KUKA KRL program: f1_Kuka_APT202T03S02.SRC

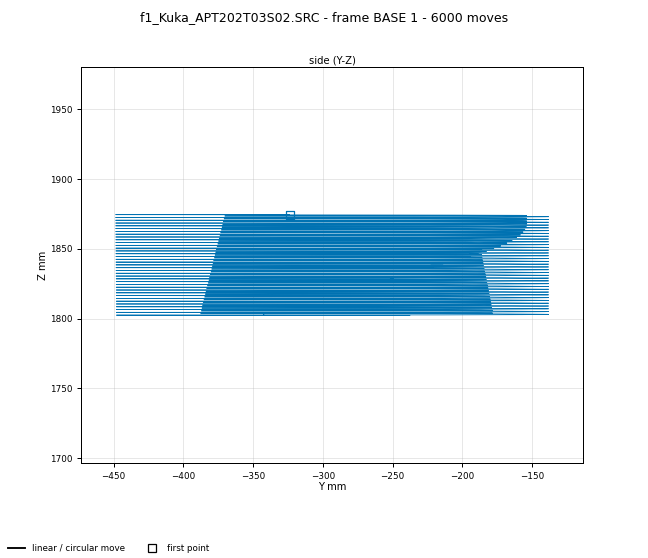
[picture p0: tool path of f1_Kuka_APT202T03S02.SRC in frame BASE 1, 6000 of 6001 moves have a stored position in this frame; points joined in program order, loops and branches not executed]
&ACCESS RVP
&REL 2
&PARAM TEMPLATE = C:\KRC\Roboter\Template\vorgabe
&PARAM EDITMASK = *
DEF f1_Kuka_APT202T03S02()


;FOLD INI;%{PE}%V3.2.0,%MKUKATPBASIS,%CINIT,%VCOMMON,%P
  ;FOLD BAS INI;%{E}%V3.2.0,%MKUKATPBASIS,%CINIT,%VINIT,%P
    GLOBAL INTERRUPT DECL 3 WHEN $STOPMESS==TRUE DO IR_STOPM ( )
    INTERRUPT ON 3
    BAS (#INITMOV,0 )
  ;ENDFOLD (BAS INI)
  ;FOLD USER INI;%{E}%V3.2.0,%MKUKATPUSER,%CINIT,%VINIT,%P
    ;Make your modifications here
  ;ENDFOLD (USER INI)
;ENDFOLD (INI)


;*** Make Null PTP Move
  PTP $pos_act

;*** Auto Load The Correct TOOL Data
  $tool=tool_data[3]

;*** Auto Load The Correct BASE Data
  $base=base_data[1]

  $ADVANCE = 5

;*** Restate Last Velocity
MMPM(30000.0)
SetRPM(6000)
LIN {X 0.160,Y -323.868,Z 1874.590,A 0.000,B 0.000,C 90.000,E1 106.260} C_DIS
LIN {X -0.109,Y -337.538,Z 1874.580,A 0.000,B 0.000,C 90.000,E1 104.411} C_DIS
LIN {X 0.038,Y -352.392,Z 1874.570,A 0.000,B 0.000,C 90.000,E1 102.535} C_DIS
LIN {X 0.047,Y -370.795,Z 1874.558,A 0.000,B 0.000,C 90.000,E1 100.489} C_DIS
LIN {X 0.119,Y -389.616,Z 1874.548,A 0.000,B 0.000,C 90.000,E1 98.624} C_DIS
LIN {X 0.014,Y -408.857,Z 1874.539,A 0.000,B 0.000,C 90.000,E1 96.947} C_DIS
LIN {X -0.177,Y -431.224,Z 1874.529,A 0.000,B 0.000,C 90.000,E1 95.220} C_DIS
LIN {X -0.017,Y -439.619,Z 1874.526,A 0.000,B 0.000,C 90.000,E1 94.588} C_DIS
LIN {X 0.199,Y -441.761,Z 1874.524,A 0.000,B 0.000,C 90.000,E1 94.359} C_DIS
LIN {X 0.089,Y -443.727,Z 1874.523,A 0.000,B 0.000,C 90.000,E1 94.131} C_DIS
LIN {X 0.009,Y -445.233,Z 1874.522,A 0.000,B 0.000,C 90.000,E1 93.898} C_DIS
LIN {X 0.189,Y -446.476,Z 1874.520,A 0.000,B 0.000,C 90.000,E1 93.612} C_DIS
LIN {X -0.075,Y -447.396,Z 1874.519,A 0.000,B 0.000,C 90.000,E1 93.383} C_DIS
LIN {X -0.118,Y -448.428,Z 1874.516,A 0.000,B 0.000,C 90.000,E1 92.865} C_DIS
LIN {X -0.177,Y -448.508,Z 1874.513,A 0.000,B 0.000,C 90.000,E1 92.350} C_DIS
LIN {X -0.213,Y -447.651,Z 1874.510,A 0.000,B 0.000,C 90.000,E1 91.833} C_DIS
LIN {X 0.183,Y -445.726,Z 1874.507,A 0.000,B 0.000,C 90.000,E1 91.260} C_DIS
LIN {X 0.128,Y -442.593,Z 1874.504,A 0.000,B 0.000,C 90.000,E1 90.745} C_DIS
LIN {X 0.008,Y -431.075,Z 1874.494,A 0.000,B 0.000,C 90.000,E1 88.912} C_DIS
LIN {X -0.023,Y -421.003,Z 1874.485,A 0.000,B 0.000,C 90.000,E1 87.306} C_DIS
LIN {X -0.120,Y -409.228,Z 1874.474,A 0.000,B 0.000,C 90.000,E1 85.412} C_DIS
LIN {X 0.015,Y -397.325,Z 1874.464,A 0.000,B 0.000,C 90.000,E1 83.451} C_DIS
LIN {X -0.090,Y -385.367,Z 1874.453,A 0.000,B 0.000,C 90.000,E1 81.489} C_DIS
LIN {X 0.040,Y -373.481,Z 1874.441,A 0.000,B 0.000,C 90.000,E1 79.454} C_DIS
LIN {X -0.066,Y -355.484,Z 1874.423,A 0.000,B 0.000,C 90.000,E1 76.228} C_DIS
LIN {X -0.066,Y -341.683,Z 1874.408,A 0.000,B 0.000,C 90.000,E1 73.504} C_DIS
LIN {X -0.122,Y -329.802,Z 1874.395,A 0.000,B 0.000,C 90.000,E1 71.040} C_DIS
LIN {X 0.107,Y -316.779,Z 1874.379,A 0.000,B 0.000,C 90.000,E1 68.156} C_DIS
LIN {X -0.103,Y -305.735,Z 1874.364,A 0.000,B 0.000,C 90.000,E1 65.613} C_DIS
LIN {X -0.074,Y -296.186,Z 1874.352,A 0.000,B 0.000,C 90.000,E1 63.307} C_DIS
LIN {X 0.124,Y -285.518,Z 1874.337,A 0.000,B 0.000,C 90.000,E1 60.589} C_DIS
LIN {X 0.126,Y -276.095,Z 1874.323,A 0.000,B 0.000,C 90.000,E1 58.201} C_DIS
LIN {X -0.021,Y -266.617,Z 1874.310,A 0.000,B 0.000,C 90.000,E1 55.801} C_DIS
LIN {X -0.060,Y -257.019,Z 1874.296,A 0.000,B 0.000,C 90.000,E1 53.336} C_DIS
LIN {X -0.008,Y -247.409,Z 1874.282,A 0.000,B 0.000,C 90.000,E1 50.803} C_DIS
LIN {X -0.043,Y -237.926,Z 1874.268,A 0.000,B 0.000,C 90.000,E1 48.243} C_DIS
LIN {X 0.069,Y -226.120,Z 1874.249,A 0.000,B 0.000,C 90.000,E1 44.838} C_DIS
LIN {X 0.023,Y -214.916,Z 1874.230,A 0.000,B 0.000,C 90.000,E1 41.391} C_DIS
LIN {X -0.011,Y -205.742,Z 1874.213,A 0.000,B 0.000,C 90.000,E1 38.257} C_DIS
LIN {X 0.104,Y -197.470,Z 1874.195,A 0.000,B 0.000,C 90.000,E1 35.025} C_DIS
LIN {X 0.003,Y -189.920,Z 1874.177,A 0.000,B 0.000,C 90.000,E1 31.799} C_DIS
LIN {X 0.010,Y -183.112,Z 1874.158,A 0.000,B 0.000,C 90.000,E1 28.487} C_DIS
LIN {X -0.080,Y -176.978,Z 1874.140,A 0.000,B 0.000,C 90.000,E1 25.155} C_DIS
LIN {X 0.016,Y -171.680,Z 1874.121,A 0.000,B 0.000,C 90.000,E1 21.716} C_DIS
LIN {X -0.053,Y -167.146,Z 1874.102,A 0.000,B 0.000,C 90.000,E1 18.290} C_DIS
LIN {X 0.038,Y -163.431,Z 1874.082,A 0.000,B 0.000,C 90.000,E1 14.773} C_DIS
LIN {X 0.056,Y -159.651,Z 1874.058,A 0.000,B 0.000,C 90.000,E1 10.366} C_DIS
LIN {X -0.049,Y -157.036,Z 1874.033,A 0.000,B 0.000,C 90.000,E1 5.967} C_DIS
LIN {X 0.000,Y -154.778,Z 1874.000,A 0.000,B 0.000,C 90.000,E1 360.000} C_DIS
LIN {X -0.018,Y -154.036,Z 1873.948,A 0.000,B 0.000,C 90.000,E1 350.557} C_DIS
LIN {X 0.044,Y -155.862,Z 1873.910,A 0.000,B 0.000,C 90.000,E1 343.866} C_DIS
LIN {X 0.028,Y -170.780,Z 1873.910,A 0.000,B 0.000,C 90.000,E1 343.866} C_DIS
LIN {X 0.085,Y -172.079,Z 1873.910,A 0.000,B 0.000,C 90.000,E1 343.740} C_DIS
LIN {X -0.020,Y -173.989,Z 1873.908,A 0.000,B 0.000,C 90.000,E1 343.378} C_DIS
LIN {X 0.067,Y -176.452,Z 1873.903,A 0.000,B 0.000,C 90.000,E1 342.489} C_DIS
LIN {X 0.060,Y -178.257,Z 1873.898,A 0.000,B 0.000,C 90.000,E1 341.638} C_DIS
LIN {X 0.074,Y -181.161,Z 1873.889,A 0.000,B 0.000,C 90.000,E1 339.934} C_DIS
LIN {X 0.059,Y -184.817,Z 1873.875,A 0.000,B 0.000,C 90.000,E1 337.411} C_DIS
LIN {X 0.007,Y -188.127,Z 1873.861,A 0.000,B 0.000,C 90.000,E1 334.921} C_DIS
LIN {X 0.086,Y -191.321,Z 1873.847,A 0.000,B 0.000,C 90.000,E1 332.410} C_DIS
LIN {X 0.054,Y -194.370,Z 1873.833,A 0.000,B 0.000,C 90.000,E1 329.950} C_DIS
LIN {X -0.030,Y -198.281,Z 1873.815,A 0.000,B 0.000,C 90.000,E1 326.707} C_DIS
LIN {X -0.010,Y -202.127,Z 1873.797,A 0.000,B 0.000,C 90.000,E1 323.463} C_DIS
LIN {X -0.041,Y -207.004,Z 1873.775,A 0.000,B 0.000,C 90.000,E1 319.461} C_DIS
LIN {X -0.015,Y -212.523,Z 1873.753,A 0.000,B 0.000,C 90.000,E1 315.486} C_DIS
LIN {X -0.044,Y -216.764,Z 1873.740,A 0.000,B 0.000,C 90.000,E1 313.137} C_DIS
LIN {X 0.048,Y -220.192,Z 1873.731,A 0.000,B 0.000,C 90.000,E1 311.553} C_DIS
LIN {X 0.099,Y -223.370,Z 1873.724,A 0.000,B 0.000,C 90.000,E1 310.378} C_DIS
LIN {X -0.028,Y -228.443,Z 1873.716,A 0.000,B 0.000,C 90.000,E1 308.874} C_DIS
LIN {X -0.060,Y -234.317,Z 1873.708,A 0.000,B 0.000,C 90.000,E1 307.363} C_DIS
LIN {X 0.011,Y -242.619,Z 1873.697,A 0.000,B 0.000,C 90.000,E1 305.471} C_DIS
LIN {X -0.115,Y -253.596,Z 1873.685,A 0.000,B 0.000,C 90.000,E1 303.293} C_DIS
LIN {X 0.003,Y -263.731,Z 1873.675,A 0.000,B 0.000,C 90.000,E1 301.465} C_DIS
LIN {X 0.085,Y -276.963,Z 1873.663,A 0.000,B 0.000,C 90.000,E1 299.333} C_DIS
LIN {X -0.007,Y -292.876,Z 1873.650,A 0.000,B 0.000,C 90.000,E1 296.950} C_DIS
LIN {X -0.031,Y -306.428,Z 1873.639,A 0.000,B 0.000,C 90.000,E1 294.951} C_DIS
LIN {X -0.111,Y -317.655,Z 1873.630,A 0.000,B 0.000,C 90.000,E1 293.334} C_DIS
LIN {X -0.060,Y -330.855,Z 1873.619,A 0.000,B 0.000,C 90.000,E1 291.408} C_DIS
LIN {X 0.139,Y -339.220,Z 1873.612,A 0.000,B 0.000,C 90.000,E1 290.120} C_DIS
LIN {X 0.001,Y -345.022,Z 1873.607,A 0.000,B 0.000,C 90.000,E1 289.214} C_DIS
LIN {X -0.077,Y -350.405,Z 1873.602,A 0.000,B 0.000,C 90.000,E1 288.308} C_DIS
LIN {X -0.111,Y -355.316,Z 1873.597,A 0.000,B 0.000,C 90.000,E1 287.402} C_DIS
LIN {X -0.098,Y -359.633,Z 1873.592,A 0.000,B 0.000,C 90.000,E1 286.496} C_DIS
LIN {X -0.151,Y -363.240,Z 1873.587,A 0.000,B 0.000,C 90.000,E1 285.607} C_DIS
LIN {X -0.132,Y -365.312,Z 1873.583,A 0.000,B 0.000,C 90.000,E1 285.009} C_DIS
LIN {X -0.103,Y -367.098,Z 1873.580,A 0.000,B 0.000,C 90.000,E1 284.411} C_DIS
LIN {X -0.157,Y -368.490,Z 1873.577,A 0.000,B 0.000,C 90.000,E1 283.828} C_DIS
LIN {X -0.113,Y -369.477,Z 1873.573,A 0.000,B 0.000,C 90.000,E1 283.231} C_DIS
LIN {X -0.146,Y -370.084,Z 1873.570,A 0.000,B 0.000,C 90.000,E1 282.647} C_DIS
LIN {X -0.172,Y -370.319,Z 1873.567,A 0.000,B 0.000,C 90.000,E1 282.063} C_DIS
LIN {X 0.171,Y -370.138,Z 1873.564,A 0.000,B 0.000,C 90.000,E1 281.422} C_DIS
LIN {X 0.152,Y -369.568,Z 1873.560,A 0.000,B 0.000,C 90.000,E1 280.838} C_DIS
LIN {X 0.132,Y -368.567,Z 1873.557,A 0.000,B 0.000,C 90.000,E1 280.254} C_DIS
LIN {X 0.108,Y -367.208,Z 1873.554,A 0.000,B 0.000,C 90.000,E1 279.670} C_DIS
LIN {X 0.017,Y -365.533,Z 1873.551,A 0.000,B 0.000,C 90.000,E1 279.095} C_DIS
LIN {X -0.049,Y -362.574,Z 1873.546,A 0.000,B 0.000,C 90.000,E1 278.219} C_DIS
LIN {X 0.160,Y -358.953,Z 1873.541,A 0.000,B 0.000,C 90.000,E1 277.296} C_DIS
LIN {X 0.027,Y -356.111,Z 1873.537,A 0.000,B 0.000,C 90.000,E1 276.720} C_DIS
LIN {X -0.118,Y -352.804,Z 1873.534,A 0.000,B 0.000,C 90.000,E1 276.144} C_DIS
LIN {X 0.069,Y -348.977,Z 1873.531,A 0.000,B 0.000,C 90.000,E1 275.511} C_DIS
LIN {X -0.112,Y -344.555,Z 1873.527,A 0.000,B 0.000,C 90.000,E1 274.935} C_DIS
LIN {X 0.025,Y -339.435,Z 1873.524,A 0.000,B 0.000,C 90.000,E1 274.302} C_DIS
LIN {X -0.150,Y -333.762,Z 1873.521,A 0.000,B 0.000,C 90.000,E1 273.726} C_DIS
LIN {X -0.082,Y -327.822,Z 1873.517,A 0.000,B 0.000,C 90.000,E1 273.151} C_DIS
LIN {X -0.081,Y -321.641,Z 1873.515,A 0.000,B 0.000,C 90.000,E1 272.636} C_DIS
LIN {X -0.035,Y -315.434,Z 1873.512,A 0.000,B 0.000,C 90.000,E1 272.178} C_DIS
LIN {X -0.091,Y -308.655,Z 1873.510,A 0.000,B 0.000,C 90.000,E1 271.776} C_DIS
LIN {X 0.135,Y -301.700,Z 1873.508,A 0.000,B 0.000,C 90.000,E1 271.375} C_DIS
LIN {X 0.052,Y -294.161,Z 1873.506,A 0.000,B 0.000,C 90.000,E1 271.088} C_DIS
LIN {X 0.005,Y -286.323,Z 1873.505,A 0.000,B 0.000,C 90.000,E1 270.859} C_DIS
LIN {X 0.062,Y -271.084,Z 1873.503,A 0.000,B 0.000,C 90.000,E1 270.516} C_DIS
LIN {X 0.002,Y -249.603,Z 1873.501,A 0.000,B 0.000,C 90.000,E1 270.115} C_DIS
LIN {X -0.117,Y -236.173,Z 1873.500,A 0.000,B 0.000,C 90.000,E1 269.943} C_DIS
LIN {X 0.022,Y -225.719,Z 1873.499,A 0.000,B 0.000,C 90.000,E1 269.828} C_DIS
LIN {X -0.002,Y -181.525,Z 1873.499,A 0.000,B 0.000,C 90.000,E1 269.828} C_DIS
LIN {X 0.040,Y -180.908,Z 1873.475,A 0.000,B 0.000,C 90.000,E1 265.527} C_DIS
LIN {X -0.082,Y -180.766,Z 1873.471,A 0.000,B 0.000,C 90.000,E1 264.723} C_DIS
LIN {X -0.011,Y -178.860,Z 1873.442,A 0.000,B 0.000,C 90.000,E1 259.634} C_DIS
LIN {X 0.061,Y -175.904,Z 1873.414,A 0.000,B 0.000,C 90.000,E1 254.519} C_DIS
LIN {X -0.001,Y -174.585,Z 1873.405,A 0.000,B 0.000,C 90.000,E1 252.834} C_DIS
LIN {X 0.034,Y -171.568,Z 1873.381,A 0.000,B 0.000,C 90.000,E1 248.539} C_DIS
LIN {X 0.016,Y -167.791,Z 1873.357,A 0.000,B 0.000,C 90.000,E1 244.229} C_DIS
LIN {X 0.030,Y -166.507,Z 1873.347,A 0.000,B 0.000,C 90.000,E1 242.487} C_DIS
LIN {X 0.026,Y -163.215,Z 1873.328,A 0.000,B 0.000,C 90.000,E1 238.997} C_DIS
LIN {X -0.009,Y -161.181,Z 1873.313,A 0.000,B 0.000,C 90.000,E1 236.373} C_DIS
LIN {X -0.010,Y -157.194,Z 1873.289,A 0.000,B 0.000,C 90.000,E1 231.949} C_DIS
LIN {X 0.037,Y -155.923,Z 1873.279,A 0.000,B 0.000,C 90.000,E1 230.150} C_DIS
LIN {X 0.093,Y -152.174,Z 1873.254,A 0.000,B 0.000,C 90.000,E1 225.648} C_DIS
LIN {X 0.002,Y -150.421,Z 1873.239,A 0.000,B 0.000,C 90.000,E1 222.975} C_DIS
LIN {X -0.072,Y -147.150,Z 1873.214,A 0.000,B 0.000,C 90.000,E1 218.463} C_DIS
LIN {X 0.015,Y -145.163,Z 1873.193,A 0.000,B 0.000,C 90.000,E1 214.771} C_DIS
LIN {X -0.069,Y -142.317,Z 1873.162,A 0.000,B 0.000,C 90.000,E1 209.283} C_DIS
LIN {X 0.051,Y -141.707,Z 1873.152,A 0.000,B 0.000,C 90.000,E1 207.385} C_DIS
LIN {X -0.025,Y -139.469,Z 1873.116,A 0.000,B 0.000,C 90.000,E1 200.918} C_DIS
LIN {X 0.028,Y -139.202,Z 1873.106,A 0.000,B 0.000,C 90.000,E1 199.033} C_DIS
LIN {X -0.045,Y -138.329,Z 1873.054,A 0.000,B 0.000,C 90.000,E1 189.726} C_DIS
LIN {X -0.042,Y -139.442,Z 1873.007,A 0.000,B 0.000,C 90.000,E1 181.318} C_DIS
LIN {X 0.037,Y -140.977,Z 1872.976,A 0.000,B 0.000,C 90.000,E1 175.698} C_DIS
LIN {X -0.013,Y -142.732,Z 1872.956,A 0.000,B 0.000,C 90.000,E1 172.008} C_DIS
LIN {X -0.056,Y -145.121,Z 1872.930,A 0.000,B 0.000,C 90.000,E1 167.409} C_DIS
LIN {X -0.061,Y -147.744,Z 1872.910,A 0.000,B 0.000,C 90.000,E1 163.740} C_DIS
LIN {X 0.021,Y -150.411,Z 1872.889,A 0.000,B 0.000,C 90.000,E1 160.061} C_DIS
LIN {X 0.035,Y -153.849,Z 1872.869,A 0.000,B 0.000,C 90.000,E1 156.433} C_DIS
LIN {X -0.048,Y -157.260,Z 1872.849,A 0.000,B 0.000,C 90.000,E1 152.871} C_DIS
LIN {X 0.031,Y -161.435,Z 1872.829,A 0.000,B 0.000,C 90.000,E1 149.282} C_DIS
LIN {X 0.038,Y -165.636,Z 1872.810,A 0.000,B 0.000,C 90.000,E1 145.754} C_DIS
LIN {X 0.020,Y -170.568,Z 1872.790,A 0.000,B 0.000,C 90.000,E1 142.271} C_DIS
LIN {X -0.072,Y -175.446,Z 1872.771,A 0.000,B 0.000,C 90.000,E1 138.852} C_DIS
LIN {X 0.044,Y -181.069,Z 1872.752,A 0.000,B 0.000,C 90.000,E1 135.405} C_DIS
LIN {X 0.034,Y -186.507,Z 1872.734,A 0.000,B 0.000,C 90.000,E1 132.043} C_DIS
LIN {X -0.023,Y -191.127,Z 1872.720,A 0.000,B 0.000,C 90.000,E1 129.564} C_DIS
LIN {X -0.103,Y -196.924,Z 1872.702,A 0.000,B 0.000,C 90.000,E1 126.297} C_DIS
LIN {X 0.091,Y -200.187,Z 1872.692,A 0.000,B 0.000,C 90.000,E1 124.612} C_DIS
LIN {X 0.088,Y -207.681,Z 1872.670,A 0.000,B 0.000,C 90.000,E1 120.590} C_DIS
LIN {X -0.011,Y -210.869,Z 1872.661,A 0.000,B 0.000,C 90.000,E1 119.027} C_DIS
LIN {X 0.099,Y -216.730,Z 1872.644,A 0.000,B 0.000,C 90.000,E1 115.848} C_DIS
LIN {X -0.081,Y -219.791,Z 1872.635,A 0.000,B 0.000,C 90.000,E1 114.335} C_DIS
LIN {X 0.027,Y -224.098,Z 1872.621,A 0.000,B 0.000,C 90.000,E1 111.844} C_DIS
LIN {X 0.002,Y -283.322,Z 1872.621,A 0.000,B 0.000,C 90.000,E1 111.844} C_DIS
LIN {X -0.099,Y -284.871,Z 1872.621,A 0.000,B 0.000,C 90.000,E1 111.844} C_DIS
LIN {X -0.061,Y -290.756,Z 1872.620,A 0.000,B 0.000,C 90.000,E1 111.535} C_DIS
LIN {X -0.022,Y -293.672,Z 1872.618,A 0.000,B 0.000,C 90.000,E1 111.227} C_DIS
LIN {X 0.150,Y -297.365,Z 1872.615,A 0.000,B 0.000,C 90.000,E1 110.610} C_DIS
LIN {X 0.073,Y -310.713,Z 1872.602,A 0.000,B 0.000,C 90.000,E1 108.308} C_DIS
LIN {X -0.103,Y -325.433,Z 1872.589,A 0.000,B 0.000,C 90.000,E1 106.079} C_DIS
LIN {X -0.029,Y -339.238,Z 1872.579,A 0.000,B 0.000,C 90.000,E1 104.175} C_DIS
LIN {X 0.156,Y -354.240,Z 1872.568,A 0.000,B 0.000,C 90.000,E1 102.299} C_DIS
LIN {X -0.051,Y -372.668,Z 1872.557,A 0.000,B 0.000,C 90.000,E1 100.310} C_DIS
LIN {X 0.047,Y -391.568,Z 1872.547,A 0.000,B 0.000,C 90.000,E1 98.454} C_DIS
LIN {X 0.079,Y -410.807,Z 1872.538,A 0.000,B 0.000,C 90.000,E1 96.777} C_DIS
LIN {X 0.013,Y -433.209,Z 1872.528,A 0.000,B 0.000,C 90.000,E1 95.049} C_DIS
LIN {X -0.010,Y -438.863,Z 1872.526,A 0.000,B 0.000,C 90.000,E1 94.645} C_DIS
LIN {X 0.200,Y -441.201,Z 1872.525,A 0.000,B 0.000,C 90.000,E1 94.416} C_DIS
LIN {X 0.217,Y -444.746,Z 1872.522,A 0.000,B 0.000,C 90.000,E1 93.955} C_DIS
LIN {X -0.055,Y -446.111,Z 1872.521,A 0.000,B 0.000,C 90.000,E1 93.726} C_DIS
LIN {X 0.118,Y -447.129,Z 1872.519,A 0.000,B 0.000,C 90.000,E1 93.440} C_DIS
LIN {X 0.075,Y -448.319,Z 1872.516,A 0.000,B 0.000,C 90.000,E1 92.922} C_DIS
LIN {X 0.014,Y -448.541,Z 1872.513,A 0.000,B 0.000,C 90.000,E1 92.407} C_DIS
LIN {X -0.037,Y -447.835,Z 1872.510,A 0.000,B 0.000,C 90.000,E1 91.892} C_DIS
LIN {X -0.073,Y -446.092,Z 1872.508,A 0.000,B 0.000,C 90.000,E1 91.375} C_DIS
LIN {X 0.123,Y -444.736,Z 1872.506,A 0.000,B 0.000,C 90.000,E1 91.088} C_DIS
LIN {X 0.201,Y -431.563,Z 1872.494,A 0.000,B 0.000,C 90.000,E1 88.969} C_DIS
LIN {X 0.175,Y -421.510,Z 1872.485,A 0.000,B 0.000,C 90.000,E1 87.364} C_DIS
LIN {X 0.083,Y -409.734,Z 1872.475,A 0.000,B 0.000,C 90.000,E1 85.469} C_DIS
LIN {X 0.180,Y -397.838,Z 1872.464,A 0.000,B 0.000,C 90.000,E1 83.514} C_DIS
LIN {X 0.125,Y -385.878,Z 1872.453,A 0.000,B 0.000,C 90.000,E1 81.546} C_DIS
LIN {X -0.107,Y -373.994,Z 1872.442,A 0.000,B 0.000,C 90.000,E1 79.567} C_DIS
LIN {X 0.081,Y -355.957,Z 1872.424,A 0.000,B 0.000,C 90.000,E1 76.297} C_DIS
LIN {X 0.173,Y -342.131,Z 1872.409,A 0.000,B 0.000,C 90.000,E1 73.559} C_DIS
LIN {X 0.124,Y -330.236,Z 1872.395,A 0.000,B 0.000,C 90.000,E1 71.094} C_DIS
LIN {X -0.052,Y -317.194,Z 1872.379,A 0.000,B 0.000,C 90.000,E1 68.284} C_DIS
LIN {X 0.156,Y -306.139,Z 1872.365,A 0.000,B 0.000,C 90.000,E1 65.665} C_DIS
LIN {X 0.058,Y -296.586,Z 1872.352,A 0.000,B 0.000,C 90.000,E1 63.384} C_DIS
LIN {X 0.007,Y -285.909,Z 1872.337,A 0.000,B 0.000,C 90.000,E1 60.717} C_DIS
LIN {X 0.022,Y -276.486,Z 1872.324,A 0.000,B 0.000,C 90.000,E1 58.329} C_DIS
LIN {X 0.111,Y -267.014,Z 1872.311,A 0.000,B 0.000,C 90.000,E1 55.881} C_DIS
LIN {X 0.073,Y -257.419,Z 1872.297,A 0.000,B 0.000,C 90.000,E1 53.417} C_DIS
LIN {X -0.066,Y -247.811,Z 1872.283,A 0.000,B 0.000,C 90.000,E1 50.928} C_DIS
LIN {X -0.104,Y -236.972,Z 1872.266,A 0.000,B 0.000,C 90.000,E1 48.000} C_DIS
LIN {X -0.009,Y -225.218,Z 1872.248,A 0.000,B 0.000,C 90.000,E1 44.595} C_DIS
LIN {X -0.081,Y -214.073,Z 1872.229,A 0.000,B 0.000,C 90.000,E1 41.148} C_DIS
LIN {X -0.024,Y -206.066,Z 1872.213,A 0.000,B 0.000,C 90.000,E1 38.382} C_DIS
LIN {X -0.020,Y -197.761,Z 1872.195,A 0.000,B 0.000,C 90.000,E1 35.185} C_DIS
LIN {X -0.002,Y -190.187,Z 1872.177,A 0.000,B 0.000,C 90.000,E1 31.926} C_DIS
LIN {X 0.010,Y -183.356,Z 1872.159,A 0.000,B 0.000,C 90.000,E1 28.615} C_DIS
LIN {X -0.075,Y -177.191,Z 1872.140,A 0.000,B 0.000,C 90.000,E1 25.283} C_DIS
LIN {X 0.027,Y -171.863,Z 1872.121,A 0.000,B 0.000,C 90.000,E1 21.844} C_DIS
LIN {X -0.035,Y -167.298,Z 1872.102,A 0.000,B 0.000,C 90.000,E1 18.417} C_DIS
LIN {X 0.062,Y -163.553,Z 1872.083,A 0.000,B 0.000,C 90.000,E1 14.898} C_DIS
LIN {X -0.067,Y -159.744,Z 1872.058,A 0.000,B 0.000,C 90.000,E1 10.546} C_DIS
LIN {X -0.005,Y -157.090,Z 1872.034,A 0.000,B 0.000,C 90.000,E1 6.087} C_DIS
LIN {X 0.000,Y -154.770,Z 1872.000,A 0.000,B 0.000,C 90.000,E1 360.000} C_DIS
LIN {X -0.019,Y -154.031,Z 1871.948,A 0.000,B 0.000,C 90.000,E1 350.557} C_DIS
LIN {X 0.073,Y -154.657,Z 1871.930,A 0.000,B 0.000,C 90.000,E1 347.409} C_DIS
LIN {X 0.061,Y -169.406,Z 1871.930,A 0.000,B 0.000,C 90.000,E1 347.409} C_DIS
LIN {X -0.015,Y -170.538,Z 1871.930,A 0.000,B 0.000,C 90.000,E1 347.353} C_DIS
LIN {X 0.060,Y -172.514,Z 1871.927,A 0.000,B 0.000,C 90.000,E1 346.937} C_DIS
LIN {X 0.015,Y -173.844,Z 1871.925,A 0.000,B 0.000,C 90.000,E1 346.520} C_DIS
LIN {X -0.072,Y -174.911,Z 1871.923,A 0.000,B 0.000,C 90.000,E1 346.117} C_DIS
LIN {X 0.027,Y -176.666,Z 1871.918,A 0.000,B 0.000,C 90.000,E1 345.227} C_DIS
LIN {X 0.083,Y -179.475,Z 1871.908,A 0.000,B 0.000,C 90.000,E1 343.504} C_DIS
LIN {X 0.055,Y -181.842,Z 1871.899,A 0.000,B 0.000,C 90.000,E1 341.819} C_DIS
LIN {X -0.078,Y -184.938,Z 1871.885,A 0.000,B 0.000,C 90.000,E1 339.337} C_DIS
LIN {X 0.043,Y -187.824,Z 1871.871,A 0.000,B 0.000,C 90.000,E1 336.794} C_DIS
LIN {X -0.068,Y -191.626,Z 1871.853,A 0.000,B 0.000,C 90.000,E1 333.512} C_DIS
LIN {X -0.095,Y -194.417,Z 1871.839,A 0.000,B 0.000,C 90.000,E1 331.051} C_DIS
LIN {X 0.058,Y -198.031,Z 1871.821,A 0.000,B 0.000,C 90.000,E1 327.740} C_DIS
LIN {X -0.046,Y -201.628,Z 1871.803,A 0.000,B 0.000,C 90.000,E1 324.529} C_DIS
LIN {X 0.017,Y -205.240,Z 1871.785,A 0.000,B 0.000,C 90.000,E1 321.295} C_DIS
LIN {X 0.026,Y -210.050,Z 1871.763,A 0.000,B 0.000,C 90.000,E1 317.310} C_DIS
LIN {X 0.105,Y -213.477,Z 1871.750,A 0.000,B 0.000,C 90.000,E1 314.919} C_DIS
LIN {X -0.011,Y -216.249,Z 1871.741,A 0.000,B 0.000,C 90.000,E1 313.380} C_DIS
LIN {X -0.028,Y -220.560,Z 1871.730,A 0.000,B 0.000,C 90.000,E1 311.434} C_DIS
LIN {X 0.049,Y -223.843,Z 1871.724,A 0.000,B 0.000,C 90.000,E1 310.253} C_DIS
LIN {X -0.072,Y -229.013,Z 1871.715,A 0.000,B 0.000,C 90.000,E1 308.749} C_DIS
LIN {X -0.096,Y -235.009,Z 1871.707,A 0.000,B 0.000,C 90.000,E1 307.237} C_DIS
LIN {X 0.135,Y -243.399,Z 1871.696,A 0.000,B 0.000,C 90.000,E1 305.311} C_DIS
LIN {X -0.115,Y -254.511,Z 1871.684,A 0.000,B 0.000,C 90.000,E1 303.166} C_DIS
LIN {X 0.015,Y -264.747,Z 1871.674,A 0.000,B 0.000,C 90.000,E1 301.337} C_DIS
LIN {X 0.119,Y -278.086,Z 1871.662,A 0.000,B 0.000,C 90.000,E1 299.205} C_DIS
LIN {X -0.044,Y -291.762,Z 1871.651,A 0.000,B 0.000,C 90.000,E1 297.180} C_DIS
LIN {X 0.172,Y -303.108,Z 1871.642,A 0.000,B 0.000,C 90.000,E1 295.463} C_DIS
LIN {X 0.168,Y -314.421,Z 1871.633,A 0.000,B 0.000,C 90.000,E1 293.823} C_DIS
LIN {X -0.077,Y -325.542,Z 1871.624,A 0.000,B 0.000,C 90.000,E1 292.259} C_DIS
LIN {X 0.047,Y -334.293,Z 1871.617,A 0.000,B 0.000,C 90.000,E1 290.972} C_DIS
LIN {X -0.147,Y -342.471,Z 1871.610,A 0.000,B 0.000,C 90.000,E1 289.758} C_DIS
LIN {X 0.089,Y -349.872,Z 1871.603,A 0.000,B 0.000,C 90.000,E1 288.489} C_DIS
LIN {X 0.052,Y -354.932,Z 1871.598,A 0.000,B 0.000,C 90.000,E1 287.583} C_DIS
LIN {X 0.065,Y -359.364,Z 1871.593,A 0.000,B 0.000,C 90.000,E1 286.677} C_DIS
LIN {X 0.012,Y -363.115,Z 1871.588,A 0.000,B 0.000,C 90.000,E1 285.788} C_DIS
LIN {X 0.030,Y -365.296,Z 1871.584,A 0.000,B 0.000,C 90.000,E1 285.190} C_DIS
LIN {X 0.061,Y -367.123,Z 1871.581,A 0.000,B 0.000,C 90.000,E1 284.592} C_DIS
LIN {X 0.008,Y -368.629,Z 1871.578,A 0.000,B 0.000,C 90.000,E1 284.008} C_DIS
LIN {X 0.054,Y -369.744,Z 1871.575,A 0.000,B 0.000,C 90.000,E1 283.411} C_DIS
LIN {X 0.023,Y -370.485,Z 1871.571,A 0.000,B 0.000,C 90.000,E1 282.827} C_DIS
LIN {X 0.000,Y -370.827,Z 1871.568,A 0.000,B 0.000,C 90.000,E1 282.243} C_DIS
LIN {X -0.016,Y -370.750,Z 1871.565,A 0.000,B 0.000,C 90.000,E1 281.658} C_DIS
LIN {X -0.030,Y -370.256,Z 1871.562,A 0.000,B 0.000,C 90.000,E1 281.074} C_DIS
LIN {X -0.046,Y -369.368,Z 1871.558,A 0.000,B 0.000,C 90.000,E1 280.489} C_DIS
LIN {X -0.064,Y -368.096,Z 1871.555,A 0.000,B 0.000,C 90.000,E1 279.905} C_DIS
LIN {X -0.090,Y -366.483,Z 1871.552,A 0.000,B 0.000,C 90.000,E1 279.321} C_DIS
LIN {X -0.181,Y -364.602,Z 1871.548,A 0.000,B 0.000,C 90.000,E1 278.746} C_DIS
LIN {X 0.103,Y -361.325,Z 1871.543,A 0.000,B 0.000,C 90.000,E1 277.814} C_DIS
LIN {X -0.056,Y -357.433,Z 1871.539,A 0.000,B 0.000,C 90.000,E1 276.947} C_DIS
LIN {X 0.157,Y -354.295,Z 1871.535,A 0.000,B 0.000,C 90.000,E1 276.315} C_DIS
LIN {X 0.000,Y -350.670,Z 1871.532,A 0.000,B 0.000,C 90.000,E1 275.739} C_DIS
LIN {X 0.172,Y -346.441,Z 1871.529,A 0.000,B 0.000,C 90.000,E1 275.106} C_DIS
LIN {X -0.024,Y -341.560,Z 1871.525,A 0.000,B 0.000,C 90.000,E1 274.531} C_DIS
LIN {X 0.092,Y -336.051,Z 1871.522,A 0.000,B 0.000,C 90.000,E1 273.898} C_DIS
LIN {X -0.008,Y -330.094,Z 1871.518,A 0.000,B 0.000,C 90.000,E1 273.326} C_DIS
LIN {X -0.137,Y -323.824,Z 1871.516,A 0.000,B 0.000,C 90.000,E1 272.808} C_DIS
LIN {X 0.043,Y -317.376,Z 1871.513,A 0.000,B 0.000,C 90.000,E1 272.293} C_DIS
LIN {X -0.065,Y -310.861,Z 1871.510,A 0.000,B 0.000,C 90.000,E1 271.892} C_DIS
LIN {X 0.097,Y -303.916,Z 1871.508,A 0.000,B 0.000,C 90.000,E1 271.489} C_DIS
LIN {X -0.053,Y -296.606,Z 1871.507,A 0.000,B 0.000,C 90.000,E1 271.203} C_DIS
LIN {X 0.131,Y -289.046,Z 1871.505,A 0.000,B 0.000,C 90.000,E1 270.917} C_DIS
LIN {X 0.002,Y -281.386,Z 1871.504,A 0.000,B 0.000,C 90.000,E1 270.745} C_DIS
LIN {X -0.103,Y -262.981,Z 1871.502,A 0.000,B 0.000,C 90.000,E1 270.401} C_DIS
LIN {X -0.096,Y -244.557,Z 1871.500,A 0.000,B 0.000,C 90.000,E1 270.057} C_DIS
LIN {X -0.042,Y -231.811,Z 1871.499,A 0.000,B 0.000,C 90.000,E1 269.885} C_DIS
LIN {X 0.044,Y -225.253,Z 1871.499,A 0.000,B 0.000,C 90.000,E1 269.828} C_DIS
LIN {X 0.013,Y -181.527,Z 1871.499,A 0.000,B 0.000,C 90.000,E1 269.828} C_DIS
LIN {X 0.040,Y -180.782,Z 1871.471,A 0.000,B 0.000,C 90.000,E1 264.723} C_DIS
LIN {X -0.065,Y -178.878,Z 1871.443,A 0.000,B 0.000,C 90.000,E1 259.690} C_DIS
LIN {X 0.011,Y -175.921,Z 1871.414,A 0.000,B 0.000,C 90.000,E1 254.574} C_DIS
LIN {X -0.099,Y -174.617,Z 1871.405,A 0.000,B 0.000,C 90.000,E1 252.906} C_DIS
LIN {X -0.007,Y -171.599,Z 1871.381,A 0.000,B 0.000,C 90.000,E1 248.592} C_DIS
LIN {X -0.018,Y -167.821,Z 1871.357,A 0.000,B 0.000,C 90.000,E1 244.280} C_DIS
LIN {X -0.001,Y -166.544,Z 1871.347,A 0.000,B 0.000,C 90.000,E1 242.538} C_DIS
LIN {X -0.090,Y -162.541,Z 1871.323,A 0.000,B 0.000,C 90.000,E1 238.201} C_DIS
LIN {X -0.030,Y -161.219,Z 1871.313,A 0.000,B 0.000,C 90.000,E1 236.421} C_DIS
LIN {X 0.005,Y -157.225,Z 1871.289,A 0.000,B 0.000,C 90.000,E1 231.984} C_DIS
LIN {X 0.029,Y -155.951,Z 1871.279,A 0.000,B 0.000,C 90.000,E1 230.194} C_DIS
LIN {X -0.013,Y -152.204,Z 1871.254,A 0.000,B 0.000,C 90.000,E1 225.729} C_DIS
LIN {X 0.008,Y -150.449,Z 1871.239,A 0.000,B 0.000,C 90.000,E1 223.014} C_DIS
LIN {X 0.035,Y -147.175,Z 1871.214,A 0.000,B 0.000,C 90.000,E1 218.463} C_DIS
LIN {X 0.002,Y -145.192,Z 1871.193,A 0.000,B 0.000,C 90.000,E1 214.818} C_DIS
LIN {X 0.037,Y -142.333,Z 1871.163,A 0.000,B 0.000,C 90.000,E1 209.283} C_DIS
LIN {X -0.034,Y -141.722,Z 1871.152,A 0.000,B 0.000,C 90.000,E1 207.462} C_DIS
LIN {X -0.052,Y -139.478,Z 1871.116,A 0.000,B 0.000,C 90.000,E1 200.972} C_DIS
LIN {X -0.063,Y -138.975,Z 1871.101,A 0.000,B 0.000,C 90.000,E1 198.181} C_DIS
LIN {X 0.059,Y -138.331,Z 1871.054,A 0.000,B 0.000,C 90.000,E1 189.726} C_DIS
LIN {X 0.062,Y -139.432,Z 1871.007,A 0.000,B 0.000,C 90.000,E1 181.318} C_DIS
LIN {X 0.002,Y -140.960,Z 1870.976,A 0.000,B 0.000,C 90.000,E1 175.755} C_DIS
LIN {X -0.048,Y -142.715,Z 1870.956,A 0.000,B 0.000,C 90.000,E1 172.064} C_DIS
LIN {X 0.052,Y -145.094,Z 1870.930,A 0.000,B 0.000,C 90.000,E1 167.409} C_DIS
LIN {X 0.047,Y -147.719,Z 1870.910,A 0.000,B 0.000,C 90.000,E1 163.740} C_DIS
LIN {X -0.011,Y -150.376,Z 1870.890,A 0.000,B 0.000,C 90.000,E1 160.115} C_DIS
LIN {X 0.006,Y -153.805,Z 1870.869,A 0.000,B 0.000,C 90.000,E1 156.485} C_DIS
LIN {X 0.066,Y -157.217,Z 1870.849,A 0.000,B 0.000,C 90.000,E1 152.871} C_DIS
LIN {X 0.006,Y -161.383,Z 1870.830,A 0.000,B 0.000,C 90.000,E1 149.331} C_DIS
LIN {X 0.017,Y -165.585,Z 1870.810,A 0.000,B 0.000,C 90.000,E1 145.801} C_DIS
LIN {X 0.004,Y -170.506,Z 1870.791,A 0.000,B 0.000,C 90.000,E1 142.316} C_DIS
LIN {X 0.048,Y -175.386,Z 1870.771,A 0.000,B 0.000,C 90.000,E1 138.852} C_DIS
LIN {X -0.089,Y -181.010,Z 1870.753,A 0.000,B 0.000,C 90.000,E1 135.486} C_DIS
LIN {X 0.035,Y -186.440,Z 1870.734,A 0.000,B 0.000,C 90.000,E1 132.081} C_DIS
LIN {X 0.104,Y -191.065,Z 1870.720,A 0.000,B 0.000,C 90.000,E1 129.564} C_DIS
LIN {X 0.026,Y -196.851,Z 1870.702,A 0.000,B 0.000,C 90.000,E1 126.297} C_DIS
LIN {X -0.056,Y -200.109,Z 1870.693,A 0.000,B 0.000,C 90.000,E1 124.692} C_DIS
LIN {X -0.063,Y -207.607,Z 1870.670,A 0.000,B 0.000,C 90.000,E1 120.669} C_DIS
LIN {X -0.061,Y -210.808,Z 1870.661,A 0.000,B 0.000,C 90.000,E1 119.077} C_DIS
LIN {X -0.055,Y -216.657,Z 1870.644,A 0.000,B 0.000,C 90.000,E1 115.924} C_DIS
LIN {X 0.056,Y -219.733,Z 1870.635,A 0.000,B 0.000,C 90.000,E1 114.335} C_DIS
LIN {X 0.032,Y -224.096,Z 1870.621,A 0.000,B 0.000,C 90.000,E1 111.844} C_DIS
LIN {X 0.005,Y -283.431,Z 1870.621,A 0.000,B 0.000,C 90.000,E1 111.844} C_DIS
LIN {X 0.054,Y -286.447,Z 1870.621,A 0.000,B 0.000,C 90.000,E1 111.770} C_DIS
LIN {X -0.082,Y -290.814,Z 1870.620,A 0.000,B 0.000,C 90.000,E1 111.535} C_DIS
LIN {X -0.114,Y -293.386,Z 1870.618,A 0.000,B 0.000,C 90.000,E1 111.280} C_DIS
LIN {X 0.091,Y -297.135,Z 1870.615,A 0.000,B 0.000,C 90.000,E1 110.663} C_DIS
LIN {X 0.001,Y -310.460,Z 1870.602,A 0.000,B 0.000,C 90.000,E1 108.362} C_DIS
LIN {X 0.125,Y -325.153,Z 1870.589,A 0.000,B 0.000,C 90.000,E1 106.079} C_DIS
LIN {X 0.120,Y -338.935,Z 1870.579,A 0.000,B 0.000,C 90.000,E1 104.189} C_DIS
LIN {X 0.047,Y -353.910,Z 1870.569,A 0.000,B 0.000,C 90.000,E1 102.355} C_DIS
LIN {X 0.174,Y -372.330,Z 1870.557,A 0.000,B 0.000,C 90.000,E1 100.310} C_DIS
LIN {X -0.125,Y -391.223,Z 1870.547,A 0.000,B 0.000,C 90.000,E1 98.511} C_DIS
LIN {X -0.123,Y -410.456,Z 1870.538,A 0.000,B 0.000,C 90.000,E1 96.834} C_DIS
LIN {X 0.208,Y -432.852,Z 1870.528,A 0.000,B 0.000,C 90.000,E1 95.049} C_DIS
LIN {X 0.183,Y -438.510,Z 1870.526,A 0.000,B 0.000,C 90.000,E1 94.645} C_DIS
LIN {X -0.047,Y -440.943,Z 1870.525,A 0.000,B 0.000,C 90.000,E1 94.473} C_DIS
LIN {X 0.060,Y -444.514,Z 1870.522,A 0.000,B 0.000,C 90.000,E1 94.012} C_DIS
LIN {X -0.213,Y -445.932,Z 1870.521,A 0.000,B 0.000,C 90.000,E1 93.784} C_DIS
LIN {X -0.040,Y -446.994,Z 1870.519,A 0.000,B 0.000,C 90.000,E1 93.498} C_DIS
LIN {X -0.086,Y -448.256,Z 1870.516,A 0.000,B 0.000,C 90.000,E1 92.980} C_DIS
LIN {X -0.148,Y -448.542,Z 1870.514,A 0.000,B 0.000,C 90.000,E1 92.465} C_DIS
LIN {X -0.199,Y -447.900,Z 1870.511,A 0.000,B 0.000,C 90.000,E1 91.949} C_DIS
LIN {X 0.210,Y -446.236,Z 1870.508,A 0.000,B 0.000,C 90.000,E1 91.375} C_DIS
LIN {X -0.039,Y -444.930,Z 1870.506,A 0.000,B 0.000,C 90.000,E1 91.146} C_DIS
LIN {X -0.105,Y -433.424,Z 1870.496,A 0.000,B 0.000,C 90.000,E1 89.312} C_DIS
LIN {X -0.090,Y -423.421,Z 1870.487,A 0.000,B 0.000,C 90.000,E1 87.707} C_DIS
LIN {X -0.136,Y -411.641,Z 1870.477,A 0.000,B 0.000,C 90.000,E1 85.812} C_DIS
LIN {X 0.019,Y -399.761,Z 1870.466,A 0.000,B 0.000,C 90.000,E1 83.856} C_DIS
LIN {X -0.043,Y -387.803,Z 1870.455,A 0.000,B 0.000,C 90.000,E1 81.894} C_DIS
LIN {X 0.143,Y -375.901,Z 1870.444,A 0.000,B 0.000,C 90.000,E1 79.859} C_DIS
LIN {X 0.030,Y -357.749,Z 1870.426,A 0.000,B 0.000,C 90.000,E1 76.645} C_DIS
LIN {X 0.096,Y -342.319,Z 1870.409,A 0.000,B 0.000,C 90.000,E1 73.614} C_DIS
LIN {X 0.059,Y -330.417,Z 1870.395,A 0.000,B 0.000,C 90.000,E1 71.148} C_DIS
LIN {X -0.050,Y -318.786,Z 1870.381,A 0.000,B 0.000,C 90.000,E1 68.646} C_DIS
LIN {X -0.011,Y -306.307,Z 1870.365,A 0.000,B 0.000,C 90.000,E1 65.741} C_DIS
LIN {X 0.028,Y -296.750,Z 1870.352,A 0.000,B 0.000,C 90.000,E1 63.435} C_DIS
LIN {X -0.153,Y -286.069,Z 1870.338,A 0.000,B 0.000,C 90.000,E1 60.795} C_DIS
LIN {X -0.131,Y -276.647,Z 1870.324,A 0.000,B 0.000,C 90.000,E1 58.408} C_DIS
LIN {X -0.037,Y -267.177,Z 1870.311,A 0.000,B 0.000,C 90.000,E1 55.960} C_DIS
LIN {X -0.070,Y -257.585,Z 1870.297,A 0.000,B 0.000,C 90.000,E1 53.497} C_DIS
LIN {X -0.009,Y -247.978,Z 1870.283,A 0.000,B 0.000,C 90.000,E1 50.964} C_DIS
LIN {X 0.104,Y -237.137,Z 1870.267,A 0.000,B 0.000,C 90.000,E1 48.000} C_DIS
LIN {X -0.126,Y -225.373,Z 1870.248,A 0.000,B 0.000,C 90.000,E1 44.676} C_DIS
LIN {X 0.115,Y -214.216,Z 1870.229,A 0.000,B 0.000,C 90.000,E1 41.148} C_DIS
LIN {X -0.123,Y -206.200,Z 1870.214,A 0.000,B 0.000,C 90.000,E1 38.463} C_DIS
LIN {X 0.006,Y -197.880,Z 1870.196,A 0.000,B 0.000,C 90.000,E1 35.231} C_DIS
LIN {X -0.081,Y -190.300,Z 1870.178,A 0.000,B 0.000,C 90.000,E1 32.005} C_DIS
LIN {X -0.060,Y -183.458,Z 1870.159,A 0.000,B 0.000,C 90.000,E1 28.693} C_DIS
LIN {X -0.061,Y -177.280,Z 1870.141,A 0.000,B 0.000,C 90.000,E1 25.335} C_DIS
LIN {X 0.040,Y -171.939,Z 1870.122,A 0.000,B 0.000,C 90.000,E1 21.897} C_DIS
LIN {X -0.025,Y -167.362,Z 1870.103,A 0.000,B 0.000,C 90.000,E1 18.471} C_DIS
LIN {X 0.071,Y -163.603,Z 1870.083,A 0.000,B 0.000,C 90.000,E1 14.954} C_DIS
LIN {X -0.060,Y -159.781,Z 1870.059,A 0.000,B 0.000,C 90.000,E1 10.602} C_DIS
LIN {X 0.001,Y -157.110,Z 1870.034,A 0.000,B 0.000,C 90.000,E1 6.144} C_DIS
LIN {X 0.000,Y -154.762,Z 1870.000,A 0.000,B 0.000,C 90.000,E1 360.000} C_DIS
LIN {X 0.053,Y -153.982,Z 1869.950,A 0.000,B 0.000,C 90.000,E1 350.971} C_DIS
LIN {X 0.038,Y -168.243,Z 1869.950,A 0.000,B 0.000,C 90.000,E1 350.971} C_DIS
LIN {X 0.069,Y -169.252,Z 1869.950,A 0.000,B 0.000,C 90.000,E1 350.905} C_DIS
LIN {X -0.021,Y -171.292,Z 1869.948,A 0.000,B 0.000,C 90.000,E1 350.557} C_DIS
LIN {X 0.065,Y -172.631,Z 1869.945,A 0.000,B 0.000,C 90.000,E1 350.095} C_DIS
LIN {X -0.020,Y -173.675,Z 1869.943,A 0.000,B 0.000,C 90.000,E1 349.690} C_DIS
LIN {X 0.032,Y -175.380,Z 1869.938,A 0.000,B 0.000,C 90.000,E1 348.814} C_DIS
LIN {X -0.012,Y -178.079,Z 1869.928,A 0.000,B 0.000,C 90.000,E1 347.117} C_DIS
LIN {X -0.021,Y -181.302,Z 1869.914,A 0.000,B 0.000,C 90.000,E1 344.574} C_DIS
LIN {X -0.044,Y -184.128,Z 1869.900,A 0.000,B 0.000,C 90.000,E1 342.054} C_DIS
LIN {X -0.075,Y -187.535,Z 1869.882,A 0.000,B 0.000,C 90.000,E1 338.720} C_DIS
LIN {X 0.073,Y -190.886,Z 1869.863,A 0.000,B 0.000,C 90.000,E1 335.357} C_DIS
LIN {X -0.057,Y -194.324,Z 1869.845,A 0.000,B 0.000,C 90.000,E1 332.103} C_DIS
LIN {X -0.007,Y -197.703,Z 1869.827,A 0.000,B 0.000,C 90.000,E1 328.820} C_DIS
LIN {X -0.071,Y -201.042,Z 1869.809,A 0.000,B 0.000,C 90.000,E1 325.595} C_DIS
LIN {X 0.014,Y -204.410,Z 1869.791,A 0.000,B 0.000,C 90.000,E1 322.351} C_DIS
LIN {X -0.010,Y -208.813,Z 1869.769,A 0.000,B 0.000,C 90.000,E1 318.366} C_DIS
LIN {X -0.014,Y -213.014,Z 1869.751,A 0.000,B 0.000,C 90.000,E1 315.202} C_DIS
LIN {X 0.016,Y -215.720,Z 1869.742,A 0.000,B 0.000,C 90.000,E1 313.623} C_DIS
LIN {X -0.067,Y -219.023,Z 1869.734,A 0.000,B 0.000,C 90.000,E1 312.081} C_DIS
LIN {X -0.030,Y -222.005,Z 1869.727,A 0.000,B 0.000,C 90.000,E1 310.906} C_DIS
LIN {X 0.061,Y -225.573,Z 1869.721,A 0.000,B 0.000,C 90.000,E1 309.725} C_DIS
LIN {X -0.040,Y -231.051,Z 1869.712,A 0.000,B 0.000,C 90.000,E1 308.222} C_DIS
LIN {X 0.121,Y -238.999,Z 1869.702,A 0.000,B 0.000,C 90.000,E1 306.297} C_DIS
LIN {X -0.070,Y -249.695,Z 1869.689,A 0.000,B 0.000,C 90.000,E1 304.119} C_DIS
LIN {X -0.021,Y -259.459,Z 1869.679,A 0.000,B 0.000,C 90.000,E1 302.291} C_DIS
LIN {X -0.030,Y -270.212,Z 1869.669,A 0.000,B 0.000,C 90.000,E1 300.512} C_DIS
LIN {X 0.035,Y -283.771,Z 1869.658,A 0.000,B 0.000,C 90.000,E1 298.409} C_DIS
LIN {X 0.104,Y -297.564,Z 1869.647,A 0.000,B 0.000,C 90.000,E1 296.360} C_DIS
LIN {X 0.038,Y -311.229,Z 1869.635,A 0.000,B 0.000,C 90.000,E1 294.387} C_DIS
LIN {X -0.030,Y -324.631,Z 1869.625,A 0.000,B 0.000,C 90.000,E1 292.461} C_DIS
LIN {X 0.057,Y -335.613,Z 1869.616,A 0.000,B 0.000,C 90.000,E1 290.865} C_DIS
LIN {X 0.000,Y -343.761,Z 1869.609,A 0.000,B 0.000,C 90.000,E1 289.631} C_DIS
LIN {X -0.092,Y -349.324,Z 1869.604,A 0.000,B 0.000,C 90.000,E1 288.725} C_DIS
LIN {X -0.139,Y -354.511,Z 1869.599,A 0.000,B 0.000,C 90.000,E1 287.819} C_DIS
LIN {X -0.134,Y -359.095,Z 1869.594,A 0.000,B 0.000,C 90.000,E1 286.913} C_DIS
LIN {X -0.194,Y -362.955,Z 1869.589,A 0.000,B 0.000,C 90.000,E1 286.024} C_DIS
LIN {X -0.177,Y -365.213,Z 1869.586,A 0.000,B 0.000,C 90.000,E1 285.426} C_DIS
LIN {X -0.147,Y -367.168,Z 1869.582,A 0.000,B 0.000,C 90.000,E1 284.828} C_DIS
LIN {X -0.204,Y -368.776,Z 1869.579,A 0.000,B 0.000,C 90.000,E1 284.245} C_DIS
LIN {X -0.158,Y -370.009,Z 1869.576,A 0.000,B 0.000,C 90.000,E1 283.647} C_DIS
LIN {X -0.188,Y -370.840,Z 1869.572,A 0.000,B 0.000,C 90.000,E1 283.063} C_DIS
LIN {X -0.209,Y -371.267,Z 1869.569,A 0.000,B 0.000,C 90.000,E1 282.479} C_DIS
LIN {X -0.147,Y -371.289,Z 1869.566,A 0.000,B 0.000,C 90.000,E1 281.883} C_DIS
LIN {X 0.202,Y -370.862,Z 1869.563,A 0.000,B 0.000,C 90.000,E1 281.243} C_DIS
LIN {X 0.188,Y -370.106,Z 1869.559,A 0.000,B 0.000,C 90.000,E1 280.658} C_DIS
LIN {X 0.170,Y -368.931,Z 1869.556,A 0.000,B 0.000,C 90.000,E1 280.074} C_DIS
LIN {X 0.086,Y -367.387,Z 1869.553,A 0.000,B 0.000,C 90.000,E1 279.500} C_DIS
LIN {X 0.056,Y -365.558,Z 1869.550,A 0.000,B 0.000,C 90.000,E1 278.916} C_DIS
LIN {X -0.063,Y -362.366,Z 1869.545,A 0.000,B 0.000,C 90.000,E1 278.049} C_DIS
LIN {X -0.127,Y -359.967,Z 1869.541,A 0.000,B 0.000,C 90.000,E1 277.466} C_DIS
LIN {X 0.014,Y -355.674,Z 1869.536,A 0.000,B 0.000,C 90.000,E1 276.549} C_DIS
LIN {X -0.095,Y -352.269,Z 1869.533,A 0.000,B 0.000,C 90.000,E1 275.967} C_DIS
LIN {X -0.024,Y -345.998,Z 1869.528,A 0.000,B 0.000,C 90.000,E1 275.049} C_DIS
LIN {X 0.119,Y -340.988,Z 1869.525,A 0.000,B 0.000,C 90.000,E1 274.416} C_DIS
LIN {X -0.049,Y -335.430,Z 1869.521,A 0.000,B 0.000,C 90.000,E1 273.841} C_DIS
LIN {X -0.055,Y -329.487,Z 1869.518,A 0.000,B 0.000,C 90.000,E1 273.269} C_DIS
LIN {X -0.109,Y -323.317,Z 1869.515,A 0.000,B 0.000,C 90.000,E1 272.751} C_DIS
LIN {X 0.099,Y -316.783,Z 1869.513,A 0.000,B 0.000,C 90.000,E1 272.236} C_DIS
LIN {X -0.020,Y -310.074,Z 1869.510,A 0.000,B 0.000,C 90.000,E1 271.835} C_DIS
LIN {X -0.136,Y -303.056,Z 1869.508,A 0.000,B 0.000,C 90.000,E1 271.489} C_DIS
LIN {X 0.060,Y -295.614,Z 1869.506,A 0.000,B 0.000,C 90.000,E1 271.146} C_DIS
LIN {X -0.007,Y -287.953,Z 1869.505,A 0.000,B 0.000,C 90.000,E1 270.917} C_DIS
LIN {X -0.099,Y -280.180,Z 1869.504,A 0.000,B 0.000,C 90.000,E1 270.745} C_DIS
LIN {X 0.063,Y -261.500,Z 1869.502,A 0.000,B 0.000,C 90.000,E1 270.344} C_DIS
LIN {X -0.120,Y -247.402,Z 1869.500,A 0.000,B 0.000,C 90.000,E1 270.115} C_DIS
LIN {X 0.024,Y -233.143,Z 1869.499,A 0.000,B 0.000,C 90.000,E1 269.885} C_DIS
LIN {X 0.078,Y -225.606,Z 1869.499,A 0.000,B 0.000,C 90.000,E1 269.828} C_DIS
LIN {X 0.040,Y -181.529,Z 1869.499,A 0.000,B 0.000,C 90.000,E1 269.828} C_DIS
LIN {X -0.018,Y -180.903,Z 1869.474,A 0.000,B 0.000,C 90.000,E1 265.298} C_DIS
LIN {X -0.068,Y -180.241,Z 1869.464,A 0.000,B 0.000,C 90.000,E1 263.628} C_DIS
LIN {X -0.049,Y -178.727,Z 1869.441,A 0.000,B 0.000,C 90.000,E1 259.398} C_DIS
LIN {X 0.018,Y -175.775,Z 1869.413,A 0.000,B 0.000,C 90.000,E1 254.283} C_DIS
LIN {X 0.007,Y -171.959,Z 1869.384,A 0.000,B 0.000,C 90.000,E1 249.156} C_DIS
LIN {X 0.044,Y -171.353,Z 1869.379,A 0.000,B 0.000,C 90.000,E1 248.284} C_DIS
LIN {X 0.021,Y -167.604,Z 1869.355,A 0.000,B 0.000,C 90.000,E1 243.973} C_DIS
LIN {X 0.034,Y -166.248,Z 1869.346,A 0.000,B 0.000,C 90.000,E1 242.231} C_DIS
LIN {X 0.022,Y -163.004,Z 1869.326,A 0.000,B 0.000,C 90.000,E1 238.742} C_DIS
LIN {X 0.068,Y -160.925,Z 1869.312,A 0.000,B 0.000,C 90.000,E1 236.087} C_DIS
LIN {X 0.045,Y -157.686,Z 1869.292,A 0.000,B 0.000,C 90.000,E1 232.557} C_DIS
LIN {X -0.016,Y -155.726,Z 1869.277,A 0.000,B 0.000,C 90.000,E1 229.908} C_DIS
LIN {X 0.037,Y -151.985,Z 1869.252,A 0.000,B 0.000,C 90.000,E1 225.405} C_DIS
LIN {X 0.053,Y -150.230,Z 1869.237,A 0.000,B 0.000,C 90.000,E1 222.690} C_DIS
LIN {X -0.023,Y -146.991,Z 1869.212,A 0.000,B 0.000,C 90.000,E1 218.177} C_DIS
LIN {X -0.033,Y -145.576,Z 1869.197,A 0.000,B 0.000,C 90.000,E1 215.438} C_DIS
LIN {X 0.084,Y -142.966,Z 1869.171,A 0.000,B 0.000,C 90.000,E1 210.797} C_DIS
LIN {X 0.014,Y -141.593,Z 1869.151,A 0.000,B 0.000,C 90.000,E1 207.129} C_DIS
LIN {X 0.061,Y -139.420,Z 1869.115,A 0.000,B 0.000,C 90.000,E1 200.610} C_DIS
LIN {X -0.018,Y -139.147,Z 1869.104,A 0.000,B 0.000,C 90.000,E1 198.779} C_DIS
LIN {X 0.004,Y -138.346,Z 1869.058,A 0.000,B 0.000,C 90.000,E1 190.366} C_DIS
LIN {X -0.011,Y -139.487,Z 1869.006,A 0.000,B 0.000,C 90.000,E1 181.031} C_DIS
LIN {X -0.071,Y -141.091,Z 1868.975,A 0.000,B 0.000,C 90.000,E1 175.469} C_DIS
LIN {X 0.023,Y -142.469,Z 1868.959,A 0.000,B 0.000,C 90.000,E1 172.648} C_DIS
LIN {X -0.029,Y -144.715,Z 1868.934,A 0.000,B 0.000,C 90.000,E1 168.049} C_DIS
LIN {X 0.064,Y -147.315,Z 1868.913,A 0.000,B 0.000,C 90.000,E1 164.338} C_DIS
LIN {X -0.063,Y -150.636,Z 1868.888,A 0.000,B 0.000,C 90.000,E1 159.826} C_DIS
LIN {X 0.013,Y -154.112,Z 1868.868,A 0.000,B 0.000,C 90.000,E1 156.177} C_DIS
LIN {X -0.064,Y -157.538,Z 1868.848,A 0.000,B 0.000,C 90.000,E1 152.615} C_DIS
LIN {X 0.102,Y -161.775,Z 1868.828,A 0.000,B 0.000,C 90.000,E1 148.997} C_DIS
LIN {X -0.014,Y -165.968,Z 1868.808,A 0.000,B 0.000,C 90.000,E1 145.515} C_DIS
LIN {X -0.019,Y -170.962,Z 1868.789,A 0.000,B 0.000,C 90.000,E1 142.029} C_DIS
LIN {X 0.033,Y -175.831,Z 1868.770,A 0.000,B 0.000,C 90.000,E1 138.566} C_DIS
LIN {X 0.028,Y -181.437,Z 1868.751,A 0.000,B 0.000,C 90.000,E1 135.162} C_DIS
LIN {X -0.098,Y -186.943,Z 1868.732,A 0.000,B 0.000,C 90.000,E1 131.838} C_DIS
LIN {X -0.100,Y -190.056,Z 1868.723,A 0.000,B 0.000,C 90.000,E1 130.172} C_DIS
LIN {X -0.085,Y -195.830,Z 1868.705,A 0.000,B 0.000,C 90.000,E1 126.870} C_DIS
LIN {X -0.017,Y -200.662,Z 1868.691,A 0.000,B 0.000,C 90.000,E1 124.405} C_DIS
LIN {X -0.001,Y -206.547,Z 1868.673,A 0.000,B 0.000,C 90.000,E1 121.180} C_DIS
LIN {X -0.014,Y -209.839,Z 1868.664,A 0.000,B 0.000,C 90.000,E1 119.589} C_DIS
LIN {X -0.089,Y -217.195,Z 1868.642,A 0.000,B 0.000,C 90.000,E1 115.668} C_DIS
LIN {X 0.064,Y -218.822,Z 1868.638,A 0.000,B 0.000,C 90.000,E1 114.847} C_DIS
LIN {X 0.030,Y -224.096,Z 1868.621,A 0.000,B 0.000,C 90.000,E1 111.844} C_DIS
LIN {X 0.003,Y -283.679,Z 1868.621,A 0.000,B 0.000,C 90.000,E1 111.844} C_DIS
LIN {X -0.103,Y -285.036,Z 1868.621,A 0.000,B 0.000,C 90.000,E1 111.844} C_DIS
LIN {X -0.016,Y -286.842,Z 1868.621,A 0.000,B 0.000,C 90.000,E1 111.770} C_DIS
LIN {X -0.113,Y -290.244,Z 1868.620,A 0.000,B 0.000,C 90.000,E1 111.589} C_DIS
LIN {X -0.110,Y -293.814,Z 1868.618,A 0.000,B 0.000,C 90.000,E1 111.227} C_DIS
LIN {X 0.108,Y -297.406,Z 1868.615,A 0.000,B 0.000,C 90.000,E1 110.610} C_DIS
LIN {X 0.030,Y -310.758,Z 1868.602,A 0.000,B 0.000,C 90.000,E1 108.308} C_DIS
LIN {X -0.146,Y -325.481,Z 1868.589,A 0.000,B 0.000,C 90.000,E1 106.079} C_DIS
LIN {X -0.072,Y -339.292,Z 1868.579,A 0.000,B 0.000,C 90.000,E1 104.175} C_DIS
LIN {X 0.111,Y -354.299,Z 1868.568,A 0.000,B 0.000,C 90.000,E1 102.299} C_DIS
LIN {X -0.095,Y -372.728,Z 1868.557,A 0.000,B 0.000,C 90.000,E1 100.310} C_DIS
LIN {X 0.006,Y -391.629,Z 1868.547,A 0.000,B 0.000,C 90.000,E1 98.454} C_DIS
LIN {X 0.039,Y -410.870,Z 1868.538,A 0.000,B 0.000,C 90.000,E1 96.777} C_DIS
LIN {X -0.025,Y -433.273,Z 1868.528,A 0.000,B 0.000,C 90.000,E1 95.049} C_DIS
LIN {X -0.047,Y -438.925,Z 1868.526,A 0.000,B 0.000,C 90.000,E1 94.645} C_DIS
LIN {X 0.163,Y -441.239,Z 1868.525,A 0.000,B 0.000,C 90.000,E1 94.416} C_DIS
LIN {X 0.155,Y -444.775,Z 1868.522,A 0.000,B 0.000,C 90.000,E1 93.955} C_DIS
LIN {X -0.117,Y -446.126,Z 1868.521,A 0.000,B 0.000,C 90.000,E1 93.726} C_DIS
LIN {X 0.056,Y -447.133,Z 1868.519,A 0.000,B 0.000,C 90.000,E1 93.440} C_DIS
LIN {X 0.012,Y -448.304,Z 1868.516,A 0.000,B 0.000,C 90.000,E1 92.922} C_DIS
LIN {X -0.049,Y -448.509,Z 1868.513,A 0.000,B 0.000,C 90.000,E1 92.407} C_DIS
LIN {X -0.100,Y -447.785,Z 1868.510,A 0.000,B 0.000,C 90.000,E1 91.892} C_DIS
LIN {X -0.135,Y -446.021,Z 1868.508,A 0.000,B 0.000,C 90.000,E1 91.375} C_DIS
LIN {X 0.060,Y -444.651,Z 1868.506,A 0.000,B 0.000,C 90.000,E1 91.088} C_DIS
LIN {X 0.139,Y -431.472,Z 1868.494,A 0.000,B 0.000,C 90.000,E1 88.969} C_DIS
LIN {X 0.112,Y -421.423,Z 1868.485,A 0.000,B 0.000,C 90.000,E1 87.364} C_DIS
LIN {X 0.021,Y -409.643,Z 1868.475,A 0.000,B 0.000,C 90.000,E1 85.469} C_DIS
LIN {X 0.117,Y -397.745,Z 1868.464,A 0.000,B 0.000,C 90.000,E1 83.514} C_DIS
LIN {X 0.063,Y -385.787,Z 1868.453,A 0.000,B 0.000,C 90.000,E1 81.546} C_DIS
LIN {X 0.199,Y -373.900,Z 1868.442,A 0.000,B 0.000,C 90.000,E1 79.511} C_DIS
LIN {X 0.018,Y -355.867,Z 1868.424,A 0.000,B 0.000,C 90.000,E1 76.297} C_DIS
LIN {X 0.110,Y -342.041,Z 1868.409,A 0.000,B 0.000,C 90.000,E1 73.559} C_DIS
LIN {X 0.061,Y -330.145,Z 1868.395,A 0.000,B 0.000,C 90.000,E1 71.094} C_DIS
LIN {X -0.115,Y -317.104,Z 1868.379,A 0.000,B 0.000,C 90.000,E1 68.284} C_DIS
LIN {X 0.094,Y -306.050,Z 1868.365,A 0.000,B 0.000,C 90.000,E1 65.665} C_DIS
LIN {X -0.004,Y -296.491,Z 1868.352,A 0.000,B 0.000,C 90.000,E1 63.384} C_DIS
LIN {X -0.056,Y -285.814,Z 1868.337,A 0.000,B 0.000,C 90.000,E1 60.717} C_DIS
LIN {X -0.039,Y -276.394,Z 1868.324,A 0.000,B 0.000,C 90.000,E1 58.329} C_DIS
LIN {X 0.049,Y -266.923,Z 1868.311,A 0.000,B 0.000,C 90.000,E1 55.881} C_DIS
LIN {X 0.011,Y -257.331,Z 1868.297,A 0.000,B 0.000,C 90.000,E1 53.417} C_DIS
LIN {X 0.066,Y -247.723,Z 1868.283,A 0.000,B 0.000,C 90.000,E1 50.884} C_DIS
LIN {X 0.012,Y -236.885,Z 1868.266,A 0.000,B 0.000,C 90.000,E1 47.957} C_DIS
LIN {X -0.070,Y -225.131,Z 1868.248,A 0.000,B 0.000,C 90.000,E1 44.595} C_DIS
LIN {X -0.140,Y -213.993,Z 1868.228,A 0.000,B 0.000,C 90.000,E1 41.148} C_DIS
LIN {X -0.084,Y -205.993,Z 1868.213,A 0.000,B 0.000,C 90.000,E1 38.382} C_DIS
LIN {X 0.036,Y -197.695,Z 1868.195,A 0.000,B 0.000,C 90.000,E1 35.152} C_DIS
LIN {X -0.059,Y -190.131,Z 1868.177,A 0.000,B 0.000,C 90.000,E1 31.926} C_DIS
LIN {X -0.047,Y -183.306,Z 1868.159,A 0.000,B 0.000,C 90.000,E1 28.615} C_DIS
LIN {X 0.104,Y -177.147,Z 1868.140,A 0.000,B 0.000,C 90.000,E1 25.207} C_DIS
LIN {X -0.029,Y -171.825,Z 1868.121,A 0.000,B 0.000,C 90.000,E1 21.844} C_DIS
LIN {X 0.069,Y -167.264,Z 1868.102,A 0.000,B 0.000,C 90.000,E1 18.362} C_DIS
LIN {X 0.008,Y -163.521,Z 1868.083,A 0.000,B 0.000,C 90.000,E1 14.898} C_DIS
LIN {X 0.036,Y -159.715,Z 1868.058,A 0.000,B 0.000,C 90.000,E1 10.489} C_DIS
LIN {X -0.059,Y -157.064,Z 1868.034,A 0.000,B 0.000,C 90.000,E1 6.087} C_DIS
LIN {X 0.000,Y -154.754,Z 1868.000,A 0.000,B 0.000,C 90.000,E1 360.000} C_DIS
LIN {X -0.015,Y -153.906,Z 1867.970,A 0.000,B 0.000,C 90.000,E1 354.546} C_DIS
LIN {X -0.037,Y -167.883,Z 1867.970,A 0.000,B 0.000,C 90.000,E1 354.546} C_DIS
LIN {X 0.048,Y -168.392,Z 1867.969,A 0.000,B 0.000,C 90.000,E1 354.489} C_DIS
LIN {X -0.008,Y -170.481,Z 1867.968,A 0.000,B 0.000,C 90.000,E1 354.147} C_DIS
LIN {X 0.076,Y -171.826,Z 1867.965,A 0.000,B 0.000,C 90.000,E1 353.685} C_DIS
LIN {X -0.011,Y -172.834,Z 1867.963,A 0.000,B 0.000,C 90.000,E1 353.280} C_DIS
LIN {X 0.008,Y -174.440,Z 1867.958,A 0.000,B 0.000,C 90.000,E1 352.413} C_DIS
LIN {X 0.068,Y -176.970,Z 1867.948,A 0.000,B 0.000,C 90.000,E1 350.679} C_DIS
LIN {X -0.077,Y -179.987,Z 1867.934,A 0.000,B 0.000,C 90.000,E1 348.173} C_DIS
LIN {X -0.094,Y -182.595,Z 1867.920,A 0.000,B 0.000,C 90.000,E1 345.644} C_DIS
LIN {X 0.028,Y -185.001,Z 1867.906,A 0.000,B 0.000,C 90.000,E1 343.087} C_DIS
LIN {X -0.046,Y -187.268,Z 1867.892,A 0.000,B 0.000,C 90.000,E1 340.604} C_DIS
LIN {X -0.044,Y -190.237,Z 1867.874,A 0.000,B 0.000,C 90.000,E1 337.283} C_DIS
LIN {X 0.078,Y -194.105,Z 1867.851,A 0.000,B 0.000,C 90.000,E1 333.127} C_DIS
LIN {X 0.033,Y -197.243,Z 1867.833,A 0.000,B 0.000,C 90.000,E1 329.871} C_DIS
LIN {X 0.021,Y -200.363,Z 1867.815,A 0.000,B 0.000,C 90.000,E1 326.628} C_DIS
LIN {X -0.026,Y -203.508,Z 1867.797,A 0.000,B 0.000,C 90.000,E1 323.417} C_DIS
LIN {X 0.108,Y -207.579,Z 1867.775,A 0.000,B 0.000,C 90.000,E1 319.380} C_DIS
LIN {X 0.075,Y -211.402,Z 1867.757,A 0.000,B 0.000,C 90.000,E1 316.215} C_DIS
LIN {X 0.027,Y -215.221,Z 1867.744,A 0.000,B 0.000,C 90.000,E1 313.866} C_DIS
LIN {X 0.086,Y -218.447,Z 1867.735,A 0.000,B 0.000,C 90.000,E1 312.285} C_DIS
LIN {X -0.027,Y -221.361,Z 1867.729,A 0.000,B 0.000,C 90.000,E1 311.148} C_DIS
LIN {X 0.137,Y -226.107,Z 1867.720,A 0.000,B 0.000,C 90.000,E1 309.564} C_DIS
LIN {X -0.048,Y -230.222,Z 1867.714,A 0.000,B 0.000,C 90.000,E1 308.463} C_DIS
LIN {X -0.089,Y -238.090,Z 1867.703,A 0.000,B 0.000,C 90.000,E1 306.583} C_DIS
LIN {X 0.045,Y -246.857,Z 1867.693,A 0.000,B 0.000,C 90.000,E1 304.692} C_DIS
LIN {X -0.141,Y -258.397,Z 1867.681,A 0.000,B 0.000,C 90.000,E1 302.546} C_DIS
LIN {X 0.057,Y -269.053,Z 1867.671,A 0.000,B 0.000,C 90.000,E1 300.718} C_DIS
LIN {X 0.107,Y -282.662,Z 1867.659,A 0.000,B 0.000,C 90.000,E1 298.615} C_DIS
LIN {X 0.042,Y -294.218,Z 1867.650,A 0.000,B 0.000,C 90.000,E1 296.924} C_DIS
LIN {X -0.093,Y -307.914,Z 1867.639,A 0.000,B 0.000,C 90.000,E1 294.951} C_DIS
LIN {X -0.152,Y -319.243,Z 1867.630,A 0.000,B 0.000,C 90.000,E1 293.334} C_DIS
LIN {X -0.071,Y -332.630,Z 1867.619,A 0.000,B 0.000,C 90.000,E1 291.408} C_DIS
LIN {X 0.151,Y -341.045,Z 1867.612,A 0.000,B 0.000,C 90.000,E1 290.120} C_DIS
LIN {X 0.030,Y -346.934,Z 1867.607,A 0.000,B 0.000,C 90.000,E1 289.214} C_DIS
LIN {X -0.030,Y -352.347,Z 1867.602,A 0.000,B 0.000,C 90.000,E1 288.308} C_DIS
LIN {X 0.028,Y -355.734,Z 1867.598,A 0.000,B 0.000,C 90.000,E1 287.692} C_DIS
LIN {X -0.065,Y -360.232,Z 1867.593,A 0.000,B 0.000,C 90.000,E1 286.804} C_DIS
LIN {X -0.006,Y -363.980,Z 1867.588,A 0.000,B 0.000,C 90.000,E1 285.898} C_DIS
LIN {X -0.017,Y -367.151,Z 1867.583,A 0.000,B 0.000,C 90.000,E1 285.009} C_DIS
LIN {X 0.019,Y -368.856,Z 1867.580,A 0.000,B 0.000,C 90.000,E1 284.411} C_DIS
LIN {X -0.025,Y -370.217,Z 1867.577,A 0.000,B 0.000,C 90.000,E1 283.828} C_DIS
LIN {X -0.054,Y -371.169,Z 1867.573,A 0.000,B 0.000,C 90.000,E1 283.244} C_DIS
LIN {X 0.008,Y -371.695,Z 1867.570,A 0.000,B 0.000,C 90.000,E1 282.647} C_DIS
LIN {X -0.007,Y -371.788,Z 1867.567,A 0.000,B 0.000,C 90.000,E1 282.063} C_DIS
LIN {X -0.017,Y -371.522,Z 1867.564,A 0.000,B 0.000,C 90.000,E1 281.478} C_DIS
LIN {X -0.027,Y -370.838,Z 1867.561,A 0.000,B 0.000,C 90.000,E1 280.894} C_DIS
LIN {X -0.039,Y -369.744,Z 1867.557,A 0.000,B 0.000,C 90.000,E1 280.310} C_DIS
LIN {X -0.057,Y -368.272,Z 1867.554,A 0.000,B 0.000,C 90.000,E1 279.726} C_DIS
LIN {X -0.141,Y -366.484,Z 1867.551,A 0.000,B 0.000,C 90.000,E1 279.151} C_DIS
LIN {X 0.163,Y -363.359,Z 1867.546,A 0.000,B 0.000,C 90.000,E1 278.219} C_DIS
LIN {X 0.020,Y -359.805,Z 1867.541,A 0.000,B 0.000,C 90.000,E1 277.352} C_DIS
LIN {X -0.158,Y -355.432,Z 1867.536,A 0.000,B 0.000,C 90.000,E1 276.486} C_DIS
LIN {X 0.044,Y -351.918,Z 1867.533,A 0.000,B 0.000,C 90.000,E1 275.853} C_DIS
LIN {X -0.124,Y -347.808,Z 1867.529,A 0.000,B 0.000,C 90.000,E1 275.277} C_DIS
LIN {X 0.031,Y -343.022,Z 1867.526,A 0.000,B 0.000,C 90.000,E1 274.645} C_DIS
LIN {X -0.151,Y -337.639,Z 1867.522,A 0.000,B 0.000,C 90.000,E1 274.069} C_DIS
LIN {X 0.114,Y -331.794,Z 1867.519,A 0.000,B 0.000,C 90.000,E1 273.440} C_DIS
LIN {X -0.029,Y -325.681,Z 1867.516,A 0.000,B 0.000,C 90.000,E1 272.922} C_DIS
LIN {X 0.068,Y -319.305,Z 1867.513,A 0.000,B 0.000,C 90.000,E1 272.407} C_DIS
LIN {X 0.151,Y -312.577,Z 1867.511,A 0.000,B 0.000,C 90.000,E1 271.949} C_DIS
LIN {X -0.068,Y -305.673,Z 1867.509,A 0.000,B 0.000,C 90.000,E1 271.604} C_DIS
LIN {X 0.022,Y -298.369,Z 1867.507,A 0.000,B 0.000,C 90.000,E1 271.260} C_DIS
LIN {X 0.143,Y -290.846,Z 1867.506,A 0.000,B 0.000,C 90.000,E1 270.974} C_DIS
LIN {X -0.033,Y -283.171,Z 1867.504,A 0.000,B 0.000,C 90.000,E1 270.802} C_DIS
LIN {X 0.131,Y -268.003,Z 1867.503,A 0.000,B 0.000,C 90.000,E1 270.458} C_DIS
LIN {X 0.080,Y -246.423,Z 1867.500,A 0.000,B 0.000,C 90.000,E1 270.057} C_DIS
LIN {X 0.002,Y -237.312,Z 1867.500,A 0.000,B 0.000,C 90.000,E1 269.943} C_DIS
LIN {X 0.112,Y -225.621,Z 1867.499,A 0.000,B 0.000,C 90.000,E1 269.828} C_DIS
LIN {X 0.070,Y -181.531,Z 1867.499,A 0.000,B 0.000,C 90.000,E1 269.828} C_DIS
LIN {X -0.050,Y -180.908,Z 1867.475,A 0.000,B 0.000,C 90.000,E1 265.584} C_DIS
LIN {X 0.008,Y -180.778,Z 1867.471,A 0.000,B 0.000,C 90.000,E1 264.723} C_DIS
LIN {X 0.078,Y -178.874,Z 1867.443,A 0.000,B 0.000,C 90.000,E1 259.634} C_DIS
LIN {X -0.021,Y -175.916,Z 1867.414,A 0.000,B 0.000,C 90.000,E1 254.574} C_DIS
LIN {X 0.034,Y -174.609,Z 1867.405,A 0.000,B 0.000,C 90.000,E1 252.851} C_DIS
LIN {X -0.039,Y -171.591,Z 1867.381,A 0.000,B 0.000,C 90.000,E1 248.592} C_DIS
LIN {X -0.050,Y -167.813,Z 1867.357,A 0.000,B 0.000,C 90.000,E1 244.280} C_DIS
LIN {X -0.032,Y -166.535,Z 1867.347,A 0.000,B 0.000,C 90.000,E1 242.538} C_DIS
LIN {X 0.017,Y -162.533,Z 1867.323,A 0.000,B 0.000,C 90.000,E1 238.152} C_DIS
LIN {X -0.061,Y -161.208,Z 1867.313,A 0.000,B 0.000,C 90.000,E1 236.421} C_DIS
LIN {X -0.024,Y -157.217,Z 1867.289,A 0.000,B 0.000,C 90.000,E1 231.984} C_DIS
LIN {X -0.002,Y -155.944,Z 1867.279,A 0.000,B 0.000,C 90.000,E1 230.194} C_DIS
LIN {X -0.042,Y -152.195,Z 1867.254,A 0.000,B 0.000,C 90.000,E1 225.729} C_DIS
LIN {X -0.021,Y -150.441,Z 1867.239,A 0.000,B 0.000,C 90.000,E1 223.014} C_DIS
LIN {X 0.007,Y -147.168,Z 1867.214,A 0.000,B 0.000,C 90.000,E1 218.463} C_DIS
LIN {X -0.027,Y -145.185,Z 1867.193,A 0.000,B 0.000,C 90.000,E1 214.818} C_DIS
LIN {X 0.008,Y -142.328,Z 1867.163,A 0.000,B 0.000,C 90.000,E1 209.283} C_DIS
LIN {X 0.003,Y -141.718,Z 1867.152,A 0.000,B 0.000,C 90.000,E1 207.436} C_DIS
LIN {X 0.051,Y -139.476,Z 1867.116,A 0.000,B 0.000,C 90.000,E1 200.918} C_DIS
LIN {X 0.042,Y -138.972,Z 1867.101,A 0.000,B 0.000,C 90.000,E1 198.127} C_DIS
LIN {X 0.030,Y -138.330,Z 1867.054,A 0.000,B 0.000,C 90.000,E1 189.726} C_DIS
LIN {X 0.034,Y -139.435,Z 1867.007,A 0.000,B 0.000,C 90.000,E1 181.318} C_DIS
LIN {X -0.026,Y -140.965,Z 1866.976,A 0.000,B 0.000,C 90.000,E1 175.755} C_DIS
LIN {X 0.064,Y -142.720,Z 1866.956,A 0.000,B 0.000,C 90.000,E1 172.008} C_DIS
LIN {X 0.023,Y -145.101,Z 1866.930,A 0.000,B 0.000,C 90.000,E1 167.409} C_DIS
LIN {X 0.018,Y -147.725,Z 1866.910,A 0.000,B 0.000,C 90.000,E1 163.740} C_DIS
LIN {X -0.041,Y -150.385,Z 1866.889,A 0.000,B 0.000,C 90.000,E1 160.115} C_DIS
LIN {X -0.024,Y -153.817,Z 1866.869,A 0.000,B 0.000,C 90.000,E1 156.485} C_DIS
LIN {X 0.035,Y -157.229,Z 1866.849,A 0.000,B 0.000,C 90.000,E1 152.871} C_DIS
LIN {X -0.024,Y -161.397,Z 1866.830,A 0.000,B 0.000,C 90.000,E1 149.331} C_DIS
LIN {X -0.013,Y -165.599,Z 1866.810,A 0.000,B 0.000,C 90.000,E1 145.801} C_DIS
LIN {X -0.027,Y -170.523,Z 1866.791,A 0.000,B 0.000,C 90.000,E1 142.316} C_DIS
LIN {X 0.016,Y -175.402,Z 1866.771,A 0.000,B 0.000,C 90.000,E1 138.852} C_DIS
LIN {X 0.007,Y -181.026,Z 1866.752,A 0.000,B 0.000,C 90.000,E1 135.445} C_DIS
LIN {X 0.001,Y -186.458,Z 1866.734,A 0.000,B 0.000,C 90.000,E1 132.081} C_DIS
LIN {X 0.070,Y -191.082,Z 1866.720,A 0.000,B 0.000,C 90.000,E1 129.564} C_DIS
LIN {X -0.009,Y -196.872,Z 1866.702,A 0.000,B 0.000,C 90.000,E1 126.297} C_DIS
LIN {X -0.091,Y -200.129,Z 1866.693,A 0.000,B 0.000,C 90.000,E1 124.692} C_DIS
LIN {X -0.100,Y -207.627,Z 1866.670,A 0.000,B 0.000,C 90.000,E1 120.669} C_DIS
LIN {X -0.097,Y -210.824,Z 1866.661,A 0.000,B 0.000,C 90.000,E1 119.077} C_DIS
LIN {X 0.004,Y -216.676,Z 1866.644,A 0.000,B 0.000,C 90.000,E1 115.899} C_DIS
LIN {X 0.019,Y -219.749,Z 1866.635,A 0.000,B 0.000,C 90.000,E1 114.335} C_DIS
LIN {X 0.049,Y -224.088,Z 1866.621,A 0.000,B 0.000,C 90.000,E1 111.844} C_DIS
LIN {X 0.029,Y -283.029,Z 1866.621,A 0.000,B 0.000,C 90.000,E1 111.844} C_DIS
LIN {X -0.084,Y -288.254,Z 1866.621,A 0.000,B 0.000,C 90.000,E1 111.716} C_DIS
LIN {X 0.070,Y -290.469,Z 1866.620,A 0.000,B 0.000,C 90.000,E1 111.535} C_DIS
LIN {X 0.111,Y -293.471,Z 1866.618,A 0.000,B 0.000,C 90.000,E1 111.227} C_DIS
LIN {X 0.074,Y -297.151,Z 1866.615,A 0.000,B 0.000,C 90.000,E1 110.663} C_DIS
LIN {X -0.016,Y -310.476,Z 1866.602,A 0.000,B 0.000,C 90.000,E1 108.362} C_DIS
LIN {X 0.107,Y -325.171,Z 1866.589,A 0.000,B 0.000,C 90.000,E1 106.079} C_DIS
LIN {X 0.102,Y -338.955,Z 1866.579,A 0.000,B 0.000,C 90.000,E1 104.189} C_DIS
LIN {X 0.027,Y -353.932,Z 1866.569,A 0.000,B 0.000,C 90.000,E1 102.355} C_DIS
LIN {X 0.156,Y -372.353,Z 1866.557,A 0.000,B 0.000,C 90.000,E1 100.310} C_DIS
LIN {X -0.141,Y -391.247,Z 1866.547,A 0.000,B 0.000,C 90.000,E1 98.511} C_DIS
LIN {X -0.139,Y -410.481,Z 1866.538,A 0.000,B 0.000,C 90.000,E1 96.834} C_DIS
LIN {X 0.193,Y -432.877,Z 1866.528,A 0.000,B 0.000,C 90.000,E1 95.049} C_DIS
LIN {X 0.168,Y -438.535,Z 1866.526,A 0.000,B 0.000,C 90.000,E1 94.645} C_DIS
LIN {X -0.063,Y -440.952,Z 1866.525,A 0.000,B 0.000,C 90.000,E1 94.473} C_DIS
LIN {X 0.031,Y -444.520,Z 1866.522,A 0.000,B 0.000,C 90.000,E1 94.012} C_DIS
LIN {X 0.202,Y -445.930,Z 1866.521,A 0.000,B 0.000,C 90.000,E1 93.726} C_DIS
LIN {X -0.071,Y -446.985,Z 1866.519,A 0.000,B 0.000,C 90.000,E1 93.498} C_DIS
LIN {X -0.115,Y -448.235,Z 1866.516,A 0.000,B 0.000,C 90.000,E1 92.980} C_DIS
LIN {X -0.178,Y -448.512,Z 1866.514,A 0.000,B 0.000,C 90.000,E1 92.465} C_DIS
LIN {X -0.230,Y -447.860,Z 1866.511,A 0.000,B 0.000,C 90.000,E1 91.949} C_DIS
LIN {X 0.181,Y -446.184,Z 1866.508,A 0.000,B 0.000,C 90.000,E1 91.375} C_DIS
LIN {X -0.069,Y -444.872,Z 1866.506,A 0.000,B 0.000,C 90.000,E1 91.146} C_DIS
LIN {X -0.135,Y -433.362,Z 1866.496,A 0.000,B 0.000,C 90.000,E1 89.312} C_DIS
LIN {X -0.121,Y -423.357,Z 1866.487,A 0.000,B 0.000,C 90.000,E1 87.707} C_DIS
LIN {X -0.167,Y -411.577,Z 1866.477,A 0.000,B 0.000,C 90.000,E1 85.812} C_DIS
LIN {X -0.013,Y -399.697,Z 1866.466,A 0.000,B 0.000,C 90.000,E1 83.856} C_DIS
LIN {X -0.075,Y -387.740,Z 1866.455,A 0.000,B 0.000,C 90.000,E1 81.894} C_DIS
LIN {X 0.111,Y -375.836,Z 1866.444,A 0.000,B 0.000,C 90.000,E1 79.859} C_DIS
LIN {X -0.003,Y -357.683,Z 1866.426,A 0.000,B 0.000,C 90.000,E1 76.645} C_DIS
LIN {X 0.064,Y -342.254,Z 1866.409,A 0.000,B 0.000,C 90.000,E1 73.614} C_DIS
LIN {X 0.025,Y -330.350,Z 1866.395,A 0.000,B 0.000,C 90.000,E1 71.148} C_DIS
LIN {X -0.085,Y -318.717,Z 1866.381,A 0.000,B 0.000,C 90.000,E1 68.646} C_DIS
LIN {X -0.045,Y -306.240,Z 1866.365,A 0.000,B 0.000,C 90.000,E1 65.741} C_DIS
LIN {X -0.008,Y -296.677,Z 1866.352,A 0.000,B 0.000,C 90.000,E1 63.435} C_DIS
LIN {X 0.061,Y -285.995,Z 1866.338,A 0.000,B 0.000,C 90.000,E1 60.745} C_DIS
LIN {X -0.023,Y -276.576,Z 1866.324,A 0.000,B 0.000,C 90.000,E1 58.377} C_DIS
LIN {X 0.075,Y -267.108,Z 1866.311,A 0.000,B 0.000,C 90.000,E1 55.928} C_DIS
LIN {X -0.106,Y -257.520,Z 1866.297,A 0.000,B 0.000,C 90.000,E1 53.497} C_DIS
LIN {X -0.046,Y -247.912,Z 1866.283,A 0.000,B 0.000,C 90.000,E1 50.964} C_DIS
LIN {X 0.067,Y -237.072,Z 1866.267,A 0.000,B 0.000,C 90.000,E1 48.000} C_DIS
LIN {X -0.004,Y -225.306,Z 1866.248,A 0.000,B 0.000,C 90.000,E1 44.636} C_DIS
LIN {X 0.079,Y -214.155,Z 1866.229,A 0.000,B 0.000,C 90.000,E1 41.148} C_DIS
LIN {X 0.002,Y -206.143,Z 1866.213,A 0.000,B 0.000,C 90.000,E1 38.418} C_DIS
LIN {X -0.031,Y -197.830,Z 1866.196,A 0.000,B 0.000,C 90.000,E1 35.231} C_DIS
LIN {X 0.044,Y -190.257,Z 1866.178,A 0.000,B 0.000,C 90.000,E1 31.957} C_DIS
LIN {X -0.096,Y -183.420,Z 1866.159,A 0.000,B 0.000,C 90.000,E1 28.693} C_DIS
LIN {X 0.064,Y -177.248,Z 1866.141,A 0.000,B 0.000,C 90.000,E1 25.283} C_DIS
LIN {X 0.004,Y -171.911,Z 1866.122,A 0.000,B 0.000,C 90.000,E1 21.897} C_DIS
LIN {X 0.099,Y -167.337,Z 1866.103,A 0.000,B 0.000,C 90.000,E1 18.417} C_DIS
LIN {X 0.036,Y -163.578,Z 1866.083,A 0.000,B 0.000,C 90.000,E1 14.954} C_DIS
LIN {X 0.062,Y -159.756,Z 1866.059,A 0.000,B 0.000,C 90.000,E1 10.546} C_DIS
LIN {X -0.034,Y -157.087,Z 1866.034,A 0.000,B 0.000,C 90.000,E1 6.144} C_DIS
LIN {X 0.000,Y -154.745,Z 1866.000,A 0.000,B 0.000,C 90.000,E1 360.000} C_DIS
LIN {X -0.051,Y -154.272,Z 1865.989,A 0.000,B 0.000,C 90.000,E1 358.108} C_DIS
LIN {X -0.077,Y -167.545,Z 1865.989,A 0.000,B 0.000,C 90.000,E1 358.108} C_DIS
LIN {X -0.081,Y -170.016,Z 1865.987,A 0.000,B 0.000,C 90.000,E1 357.764} C_DIS
LIN {X -0.012,Y -171.367,Z 1865.985,A 0.000,B 0.000,C 90.000,E1 357.306} C_DIS
LIN {X 0.058,Y -172.372,Z 1865.983,A 0.000,B 0.000,C 90.000,E1 356.849} C_DIS
LIN {X 0.056,Y -173.943,Z 1865.978,A 0.000,B 0.000,C 90.000,E1 355.988} C_DIS
LIN {X -0.087,Y -176.289,Z 1865.968,A 0.000,B 0.000,C 90.000,E1 354.318} C_DIS
LIN {X -0.023,Y -178.157,Z 1865.959,A 0.000,B 0.000,C 90.000,E1 352.591} C_DIS
LIN {X 0.000,Y -180.626,Z 1865.945,A 0.000,B 0.000,C 90.000,E1 350.038} C_DIS
LIN {X -0.041,Y -182.868,Z 1865.931,A 0.000,B 0.000,C 90.000,E1 347.521} C_DIS
LIN {X -0.010,Y -185.654,Z 1865.912,A 0.000,B 0.000,C 90.000,E1 344.157} C_DIS
LIN {X 0.049,Y -187.683,Z 1865.898,A 0.000,B 0.000,C 90.000,E1 341.638} C_DIS
LIN {X -0.007,Y -190.305,Z 1865.880,A 0.000,B 0.000,C 90.000,E1 338.337} C_DIS
LIN {X 0.039,Y -193.775,Z 1865.857,A 0.000,B 0.000,C 90.000,E1 334.204} C_DIS
LIN {X 0.069,Y -196.694,Z 1865.839,A 0.000,B 0.000,C 90.000,E1 330.923} C_DIS
LIN {X -0.059,Y -199.590,Z 1865.821,A 0.000,B 0.000,C 90.000,E1 327.709} C_DIS
LIN {X -0.072,Y -202.528,Z 1865.803,A 0.000,B 0.000,C 90.000,E1 324.482} C_DIS
LIN {X 0.061,Y -206.337,Z 1865.780,A 0.000,B 0.000,C 90.000,E1 320.436} C_DIS
LIN {X 0.076,Y -210.958,Z 1865.758,A 0.000,B 0.000,C 90.000,E1 316.458} C_DIS
LIN {X 0.019,Y -214.756,Z 1865.745,A 0.000,B 0.000,C 90.000,E1 314.109} C_DIS
LIN {X 0.073,Y -217.906,Z 1865.736,A 0.000,B 0.000,C 90.000,E1 312.528} C_DIS
LIN {X -0.045,Y -220.733,Z 1865.730,A 0.000,B 0.000,C 90.000,E1 311.391} C_DIS
LIN {X 0.009,Y -224.132,Z 1865.723,A 0.000,B 0.000,C 90.000,E1 310.216} C_DIS
LIN {X -0.016,Y -228.011,Z 1865.717,A 0.000,B 0.000,C 90.000,E1 309.072} C_DIS
LIN {X 0.096,Y -233.972,Z 1865.709,A 0.000,B 0.000,C 90.000,E1 307.523} C_DIS
LIN {X -0.028,Y -242.301,Z 1865.698,A 0.000,B 0.000,C 90.000,E1 305.678} C_DIS
LIN {X 0.063,Y -255.383,Z 1865.684,A 0.000,B 0.000,C 90.000,E1 303.086} C_DIS
LIN {X -0.153,Y -265.721,Z 1865.674,A 0.000,B 0.000,C 90.000,E1 301.337} C_DIS
LIN {X -0.037,Y -279.291,Z 1865.662,A 0.000,B 0.000,C 90.000,E1 299.205} C_DIS
LIN {X 0.077,Y -293.174,Z 1865.651,A 0.000,B 0.000,C 90.000,E1 297.129} C_DIS
LIN {X -0.072,Y -306.926,Z 1865.640,A 0.000,B 0.000,C 90.000,E1 295.155} C_DIS
LIN {X 0.065,Y -316.078,Z 1865.632,A 0.000,B 0.000,C 90.000,E1 293.823} C_DIS
LIN {X 0.144,Y -327.300,Z 1865.624,A 0.000,B 0.000,C 90.000,E1 292.206} C_DIS
LIN {X -0.012,Y -336.136,Z 1865.616,A 0.000,B 0.000,C 90.000,E1 290.972} C_DIS
LIN {X -0.185,Y -344.379,Z 1865.610,A 0.000,B 0.000,C 90.000,E1 289.758} C_DIS
LIN {X 0.164,Y -350.060,Z 1865.604,A 0.000,B 0.000,C 90.000,E1 288.779} C_DIS
LIN {X 0.132,Y -355.298,Z 1865.599,A 0.000,B 0.000,C 90.000,E1 287.873} C_DIS
LIN {X 0.036,Y -359.957,Z 1865.594,A 0.000,B 0.000,C 90.000,E1 286.985} C_DIS
LIN {X 0.094,Y -363.881,Z 1865.589,A 0.000,B 0.000,C 90.000,E1 286.079} C_DIS
LIN {X 0.084,Y -367.148,Z 1865.584,A 0.000,B 0.000,C 90.000,E1 285.190} C_DIS
LIN {X 0.127,Y -368.926,Z 1865.581,A 0.000,B 0.000,C 90.000,E1 284.592} C_DIS
LIN {X 0.084,Y -370.376,Z 1865.578,A 0.000,B 0.000,C 90.000,E1 284.008} C_DIS
LIN {X 0.142,Y -371.445,Z 1865.575,A 0.000,B 0.000,C 90.000,E1 283.411} C_DIS
LIN {X 0.122,Y -372.097,Z 1865.571,A 0.000,B 0.000,C 90.000,E1 282.827} C_DIS
LIN {X 0.110,Y -372.325,Z 1865.568,A 0.000,B 0.000,C 90.000,E1 282.243} C_DIS
LIN {X 0.103,Y -372.154,Z 1865.565,A 0.000,B 0.000,C 90.000,E1 281.658} C_DIS
LIN {X 0.097,Y -371.531,Z 1865.562,A 0.000,B 0.000,C 90.000,E1 281.074} C_DIS
LIN {X 0.091,Y -370.495,Z 1865.558,A 0.000,B 0.000,C 90.000,E1 280.489} C_DIS
LIN {X 0.080,Y -369.148,Z 1865.555,A 0.000,B 0.000,C 90.000,E1 279.905} C_DIS
LIN {X 0.059,Y -367.412,Z 1865.552,A 0.000,B 0.000,C 90.000,E1 279.321} C_DIS
LIN {X -0.066,Y -363.200,Z 1865.545,A 0.000,B 0.000,C 90.000,E1 278.163} C_DIS
LIN {X 0.150,Y -359.607,Z 1865.540,A 0.000,B 0.000,C 90.000,E1 277.239} C_DIS
LIN {X -0.025,Y -355.179,Z 1865.535,A 0.000,B 0.000,C 90.000,E1 276.372} C_DIS
LIN {X 0.174,Y -351.536,Z 1865.532,A 0.000,B 0.000,C 90.000,E1 275.739} C_DIS
LIN {X 0.004,Y -347.335,Z 1865.529,A 0.000,B 0.000,C 90.000,E1 275.163} C_DIS
LIN {X 0.155,Y -342.428,Z 1865.525,A 0.000,B 0.000,C 90.000,E1 274.531} C_DIS
LIN {X -0.062,Y -336.855,Z 1865.522,A 0.000,B 0.000,C 90.000,E1 273.955} C_DIS
LIN {X -0.096,Y -330.930,Z 1865.519,A 0.000,B 0.000,C 90.000,E1 273.383} C_DIS
LIN {X -0.147,Y -324.863,Z 1865.516,A 0.000,B 0.000,C 90.000,E1 272.865} C_DIS
LIN {X 0.049,Y -318.485,Z 1865.513,A 0.000,B 0.000,C 90.000,E1 272.350} C_DIS
LIN {X -0.080,Y -311.949,Z 1865.511,A 0.000,B 0.000,C 90.000,E1 271.949} C_DIS
LIN {X 0.060,Y -305.072,Z 1865.509,A 0.000,B 0.000,C 90.000,E1 271.547} C_DIS
LIN {X -0.143,Y -297.611,Z 1865.507,A 0.000,B 0.000,C 90.000,E1 271.260} C_DIS
LIN {X 0.013,Y -289.916,Z 1865.505,A 0.000,B 0.000,C 90.000,E1 270.974} C_DIS
LIN {X -0.140,Y -282.081,Z 1865.504,A 0.000,B 0.000,C 90.000,E1 270.802} C_DIS
LIN {X 0.070,Y -267.051,Z 1865.503,A 0.000,B 0.000,C 90.000,E1 270.458} C_DIS
LIN {X 0.047,Y -245.442,Z 1865.500,A 0.000,B 0.000,C 90.000,E1 270.057} C_DIS
LIN {X -0.031,Y -236.173,Z 1865.500,A 0.000,B 0.000,C 90.000,E1 269.943} C_DIS
LIN {X -0.095,Y -225.842,Z 1865.499,A 0.000,B 0.000,C 90.000,E1 269.885} C_DIS
LIN {X 0.082,Y -181.532,Z 1865.499,A 0.000,B 0.000,C 90.000,E1 269.828} C_DIS
LIN {X -0.053,Y -180.792,Z 1865.471,A 0.000,B 0.000,C 90.000,E1 264.780} C_DIS
LIN {X 0.022,Y -178.890,Z 1865.443,A 0.000,B 0.000,C 90.000,E1 259.690} C_DIS
LIN {X -0.072,Y -175.933,Z 1865.414,A 0.000,B 0.000,C 90.000,E1 254.629} C_DIS
LIN {X 0.043,Y -175.380,Z 1865.410,A 0.000,B 0.000,C 90.000,E1 253.740} C_DIS
LIN {X 0.040,Y -172.154,Z 1865.386,A 0.000,B 0.000,C 90.000,E1 249.464} C_DIS
LIN {X 0.078,Y -171.619,Z 1865.381,A 0.000,B 0.000,C 90.000,E1 248.592} C_DIS
LIN {X 0.066,Y -167.843,Z 1865.357,A 0.000,B 0.000,C 90.000,E1 244.280} C_DIS
LIN {X 0.005,Y -166.571,Z 1865.348,A 0.000,B 0.000,C 90.000,E1 242.564} C_DIS
LIN {X -0.008,Y -162.564,Z 1865.323,A 0.000,B 0.000,C 90.000,E1 238.201} C_DIS
LIN {X 0.052,Y -161.244,Z 1865.314,A 0.000,B 0.000,C 90.000,E1 236.421} C_DIS
LIN {X -0.038,Y -157.247,Z 1865.289,A 0.000,B 0.000,C 90.000,E1 232.029} C_DIS
LIN {X 0.009,Y -155.970,Z 1865.279,A 0.000,B 0.000,C 90.000,E1 230.231} C_DIS
LIN {X 0.066,Y -152.225,Z 1865.254,A 0.000,B 0.000,C 90.000,E1 225.729} C_DIS
LIN {X -0.023,Y -150.468,Z 1865.239,A 0.000,B 0.000,C 90.000,E1 223.056} C_DIS
LIN {X -0.003,Y -147.193,Z 1865.214,A 0.000,B 0.000,C 90.000,E1 218.508} C_DIS
LIN {X 0.079,Y -145.212,Z 1865.194,A 0.000,B 0.000,C 90.000,E1 214.818} C_DIS
LIN {X -0.012,Y -142.344,Z 1865.163,A 0.000,B 0.000,C 90.000,E1 209.333} C_DIS
LIN {X 0.042,Y -141.732,Z 1865.153,A 0.000,B 0.000,C 90.000,E1 207.462} C_DIS
LIN {X 0.023,Y -139.483,Z 1865.117,A 0.000,B 0.000,C 90.000,E1 200.972} C_DIS
LIN {X 0.011,Y -138.983,Z 1865.101,A 0.000,B 0.000,C 90.000,E1 198.181} C_DIS
LIN {X -0.027,Y -138.334,Z 1865.054,A 0.000,B 0.000,C 90.000,E1 189.792} C_DIS
LIN {X -0.003,Y -139.425,Z 1865.008,A 0.000,B 0.000,C 90.000,E1 181.375} C_DIS
LIN {X 0.051,Y -141.349,Z 1864.971,A 0.000,B 0.000,C 90.000,E1 174.837} C_DIS
LIN {X 0.028,Y -142.704,Z 1864.956,A 0.000,B 0.000,C 90.000,E1 172.064} C_DIS
LIN {X -0.013,Y -145.074,Z 1864.930,A 0.000,B 0.000,C 90.000,E1 167.465} C_DIS
LIN {X -0.017,Y -147.699,Z 1864.910,A 0.000,B 0.000,C 90.000,E1 163.795} C_DIS
LIN {X 0.016,Y -150.351,Z 1864.890,A 0.000,B 0.000,C 90.000,E1 160.134} C_DIS
LIN {X 0.009,Y -154.606,Z 1864.865,A 0.000,B 0.000,C 90.000,E1 155.613} C_DIS
LIN {X 0.016,Y -158.147,Z 1864.845,A 0.000,B 0.000,C 90.000,E1 152.025} C_DIS
LIN {X 0.060,Y -162.434,Z 1864.825,A 0.000,B 0.000,C 90.000,E1 148.456} C_DIS
LIN {X -0.044,Y -166.693,Z 1864.805,A 0.000,B 0.000,C 90.000,E1 144.975} C_DIS
LIN {X 0.068,Y -171.698,Z 1864.786,A 0.000,B 0.000,C 90.000,E1 141.457} C_DIS
LIN {X 0.003,Y -176.672,Z 1864.767,A 0.000,B 0.000,C 90.000,E1 138.038} C_DIS
LIN {X -0.001,Y -180.968,Z 1864.753,A 0.000,B 0.000,C 90.000,E1 135.486} C_DIS
LIN {X -0.014,Y -186.391,Z 1864.734,A 0.000,B 0.000,C 90.000,E1 132.123} C_DIS
LIN {X -0.074,Y -191.020,Z 1864.720,A 0.000,B 0.000,C 90.000,E1 129.644} C_DIS
LIN {X 0.118,Y -196.800,Z 1864.702,A 0.000,B 0.000,C 90.000,E1 126.297} C_DIS
LIN {X 0.037,Y -200.053,Z 1864.693,A 0.000,B 0.000,C 90.000,E1 124.692} C_DIS
LIN {X 0.031,Y -207.554,Z 1864.670,A 0.000,B 0.000,C 90.000,E1 120.669} C_DIS
LIN {X 0.035,Y -210.764,Z 1864.662,A 0.000,B 0.000,C 90.000,E1 119.077} C_DIS
LIN {X 0.043,Y -216.605,Z 1864.644,A 0.000,B 0.000,C 90.000,E1 115.924} C_DIS
LIN {X -0.046,Y -219.691,Z 1864.635,A 0.000,B 0.000,C 90.000,E1 114.387} C_DIS
LIN {X 0.046,Y -224.089,Z 1864.621,A 0.000,B 0.000,C 90.000,E1 111.844} C_DIS
LIN {X 0.027,Y -283.420,Z 1864.621,A 0.000,B 0.000,C 90.000,E1 111.844} C_DIS
LIN {X 0.073,Y -285.808,Z 1864.621,A 0.000,B 0.000,C 90.000,E1 111.791} C_DIS
LIN {X 0.046,Y -290.538,Z 1864.620,A 0.000,B 0.000,C 90.000,E1 111.535} C_DIS
LIN {X 0.016,Y -293.183,Z 1864.618,A 0.000,B 0.000,C 90.000,E1 111.280} C_DIS
LIN {X -0.095,Y -296.926,Z 1864.615,A 0.000,B 0.000,C 90.000,E1 110.737} C_DIS
LIN {X -0.093,Y -310.229,Z 1864.602,A 0.000,B 0.000,C 90.000,E1 108.417} C_DIS
LIN {X 0.018,Y -324.899,Z 1864.590,A 0.000,B 0.000,C 90.000,E1 106.134} C_DIS
LIN {X 0.001,Y -338.660,Z 1864.579,A 0.000,B 0.000,C 90.000,E1 104.245} C_DIS
LIN {X -0.087,Y -353.612,Z 1864.569,A 0.000,B 0.000,C 90.000,E1 102.411} C_DIS
LIN {X 0.011,Y -372.022,Z 1864.558,A 0.000,B 0.000,C 90.000,E1 100.366} C_DIS
LIN {X 0.070,Y -390.908,Z 1864.547,A 0.000,B 0.000,C 90.000,E1 98.511} C_DIS
LIN {X 0.063,Y -410.136,Z 1864.538,A 0.000,B 0.000,C 90.000,E1 96.834} C_DIS
LIN {X -0.046,Y -432.527,Z 1864.528,A 0.000,B 0.000,C 90.000,E1 95.106} C_DIS
LIN {X -0.079,Y -438.184,Z 1864.526,A 0.000,B 0.000,C 90.000,E1 94.702} C_DIS
LIN {X 0.126,Y -440.691,Z 1864.525,A 0.000,B 0.000,C 90.000,E1 94.473} C_DIS
LIN {X -0.137,Y -444.289,Z 1864.522,A 0.000,B 0.000,C 90.000,E1 94.069} C_DIS
LIN {X 0.033,Y -445.753,Z 1864.521,A 0.000,B 0.000,C 90.000,E1 93.784} C_DIS
LIN {X 0.205,Y -446.851,Z 1864.520,A 0.000,B 0.000,C 90.000,E1 93.498} C_DIS
LIN {X 0.160,Y -448.170,Z 1864.517,A 0.000,B 0.000,C 90.000,E1 92.980} C_DIS
LIN {X 0.096,Y -448.508,Z 1864.514,A 0.000,B 0.000,C 90.000,E1 92.465} C_DIS
LIN {X 0.043,Y -447.919,Z 1864.511,A 0.000,B 0.000,C 90.000,E1 91.949} C_DIS
LIN {X 0.008,Y -446.317,Z 1864.508,A 0.000,B 0.000,C 90.000,E1 91.432} C_DIS
LIN {X 0.203,Y -445.052,Z 1864.506,A 0.000,B 0.000,C 90.000,E1 91.146} C_DIS
LIN {X 0.133,Y -433.566,Z 1864.496,A 0.000,B 0.000,C 90.000,E1 89.312} C_DIS
LIN {X 0.144,Y -423.566,Z 1864.487,A 0.000,B 0.000,C 90.000,E1 87.707} C_DIS
LIN {X 0.095,Y -411.783,Z 1864.477,A 0.000,B 0.000,C 90.000,E1 85.812} C_DIS
LIN {X -0.151,Y -399.906,Z 1864.466,A 0.000,B 0.000,C 90.000,E1 83.913} C_DIS
LIN {X 0.181,Y -387.949,Z 1864.455,A 0.000,B 0.000,C 90.000,E1 81.894} C_DIS
LIN {X -0.073,Y -376.043,Z 1864.444,A 0.000,B 0.000,C 90.000,E1 79.926} C_DIS
LIN {X -0.105,Y -357.874,Z 1864.426,A 0.000,B 0.000,C 90.000,E1 76.700} C_DIS
LIN {X -0.120,Y -342.433,Z 1864.409,A 0.000,B 0.000,C 90.000,E1 73.685} C_DIS
LIN {X -0.157,Y -330.523,Z 1864.396,A 0.000,B 0.000,C 90.000,E1 71.221} C_DIS
LIN {X 0.032,Y -318.885,Z 1864.381,A 0.000,B 0.000,C 90.000,E1 68.666} C_DIS
LIN {X -0.096,Y -306.397,Z 1864.365,A 0.000,B 0.000,C 90.000,E1 65.793} C_DIS
LIN {X 0.084,Y -296.833,Z 1864.353,A 0.000,B 0.000,C 90.000,E1 63.461} C_DIS
LIN {X 0.031,Y -286.149,Z 1864.338,A 0.000,B 0.000,C 90.000,E1 60.795} C_DIS
LIN {X 0.048,Y -276.728,Z 1864.325,A 0.000,B 0.000,C 90.000,E1 58.408} C_DIS
LIN {X -0.083,Y -267.264,Z 1864.311,A 0.000,B 0.000,C 90.000,E1 56.008} C_DIS
LIN {X 0.101,Y -257.680,Z 1864.297,A 0.000,B 0.000,C 90.000,E1 53.497} C_DIS
LIN {X -0.034,Y -248.072,Z 1864.283,A 0.000,B 0.000,C 90.000,E1 51.009} C_DIS
LIN {X -0.068,Y -237.229,Z 1864.267,A 0.000,B 0.000,C 90.000,E1 48.081} C_DIS
LIN {X 0.030,Y -225.454,Z 1864.248,A 0.000,B 0.000,C 90.000,E1 44.676} C_DIS
LIN {X -0.036,Y -214.291,Z 1864.229,A 0.000,B 0.000,C 90.000,E1 41.229} C_DIS
LIN {X 0.024,Y -206.269,Z 1864.214,A 0.000,B 0.000,C 90.000,E1 38.463} C_DIS
LIN {X 0.034,Y -197.946,Z 1864.196,A 0.000,B 0.000,C 90.000,E1 35.264} C_DIS
LIN {X 0.057,Y -190.365,Z 1864.178,A 0.000,B 0.000,C 90.000,E1 32.005} C_DIS
LIN {X 0.075,Y -183.516,Z 1864.160,A 0.000,B 0.000,C 90.000,E1 28.693} C_DIS
LIN {X 0.071,Y -177.334,Z 1864.141,A 0.000,B 0.000,C 90.000,E1 25.335} C_DIS
LIN {X -0.055,Y -171.985,Z 1864.122,A 0.000,B 0.000,C 90.000,E1 21.972} C_DIS
LIN {X 0.049,Y -167.397,Z 1864.103,A 0.000,B 0.000,C 90.000,E1 18.489} C_DIS
LIN {X 0.038,Y -163.625,Z 1864.083,A 0.000,B 0.000,C 90.000,E1 15.009} C_DIS
LIN {X 0.063,Y -159.791,Z 1864.059,A 0.000,B 0.000,C 90.000,E1 10.602} C_DIS
LIN {X -0.034,Y -157.105,Z 1864.034,A 0.000,B 0.000,C 90.000,E1 6.201} C_DIS
LIN {X 0.060,Y -155.259,Z 1864.009,A 0.000,B 0.000,C 90.000,E1 1.604} C_DIS
LIN {X 0.036,Y -167.735,Z 1864.009,A 0.000,B 0.000,C 90.000,E1 1.604} C_DIS
LIN {X 0.059,Y -168.593,Z 1864.009,A 0.000,B 0.000,C 90.000,E1 1.547} C_DIS
LIN {X -0.073,Y -169.643,Z 1864.008,A 0.000,B 0.000,C 90.000,E1 1.432} C_DIS
LIN {X 0.086,Y -171.537,Z 1864.005,A 0.000,B 0.000,C 90.000,E1 0.802} C_DIS
LIN {X 0.000,Y -173.195,Z 1864.000,A 0.000,B 0.000,C 90.000,E1 360.000} C_DIS
LIN {X -0.028,Y -175.072,Z 1863.993,A 0.000,B 0.000,C 90.000,E1 358.682} C_DIS
LIN {X -0.003,Y -176.934,Z 1863.983,A 0.000,B 0.000,C 90.000,E1 356.963} C_DIS
LIN {X -0.070,Y -179.252,Z 1863.969,A 0.000,B 0.000,C 90.000,E1 354.432} C_DIS
LIN {X -0.073,Y -181.241,Z 1863.955,A 0.000,B 0.000,C 90.000,E1 351.894} C_DIS
LIN {X 0.008,Y -183.135,Z 1863.941,A 0.000,B 0.000,C 90.000,E1 349.342} C_DIS
LIN {X 0.002,Y -185.586,Z 1863.922,A 0.000,B 0.000,C 90.000,E1 345.992} C_DIS
LIN {X -0.038,Y -187.984,Z 1863.904,A 0.000,B 0.000,C 90.000,E1 342.670} C_DIS
LIN {X 0.020,Y -190.337,Z 1863.885,A 0.000,B 0.000,C 90.000,E1 339.337} C_DIS
LIN {X -0.020,Y -193.422,Z 1863.862,A 0.000,B 0.000,C 90.000,E1 335.229} C_DIS
LIN {X -0.092,Y -196.116,Z 1863.844,A 0.000,B 0.000,C 90.000,E1 331.975} C_DIS
LIN {X 0.104,Y -198.823,Z 1863.826,A 0.000,B 0.000,C 90.000,E1 328.663} C_DIS
LIN {X -0.039,Y -201.536,Z 1863.808,A 0.000,B 0.000,C 90.000,E1 325.468} C_DIS
LIN {X -0.063,Y -205.184,Z 1863.786,A 0.000,B 0.000,C 90.000,E1 321.457} C_DIS
LIN {X -0.065,Y -209.558,Z 1863.764,A 0.000,B 0.000,C 90.000,E1 317.472} C_DIS
LIN {X 0.003,Y -213.003,Z 1863.750,A 0.000,B 0.000,C 90.000,E1 315.081} C_DIS
LIN {X 0.036,Y -215.854,Z 1863.742,A 0.000,B 0.000,C 90.000,E1 313.500} C_DIS
LIN {X 0.020,Y -220.297,Z 1863.731,A 0.000,B 0.000,C 90.000,E1 311.553} C_DIS
LIN {X 0.072,Y -223.623,Z 1863.724,A 0.000,B 0.000,C 90.000,E1 310.378} C_DIS
LIN {X 0.125,Y -228.844,Z 1863.716,A 0.000,B 0.000,C 90.000,E1 308.830} C_DIS
LIN {X 0.068,Y -236.571,Z 1863.705,A 0.000,B 0.000,C 90.000,E1 306.950} C_DIS
LIN {X -0.016,Y -245.223,Z 1863.695,A 0.000,B 0.000,C 90.000,E1 305.105} C_DIS
LIN {X 0.118,Y -256.666,Z 1863.683,A 0.000,B 0.000,C 90.000,E1 302.880} C_DIS
LIN {X -0.070,Y -267.146,Z 1863.673,A 0.000,B 0.000,C 90.000,E1 301.131} C_DIS
LIN {X -0.059,Y -280.819,Z 1863.661,A 0.000,B 0.000,C 90.000,E1 299.027} C_DIS
LIN {X 0.090,Y -294.737,Z 1863.650,A 0.000,B 0.000,C 90.000,E1 296.950} C_DIS
LIN {X 0.108,Y -308.579,Z 1863.639,A 0.000,B 0.000,C 90.000,E1 294.951} C_DIS
LIN {X 0.059,Y -319.988,Z 1863.630,A 0.000,B 0.000,C 90.000,E1 293.334} C_DIS
LIN {X 0.165,Y -333.479,Z 1863.619,A 0.000,B 0.000,C 90.000,E1 291.408} C_DIS
LIN {X 0.083,Y -341.976,Z 1863.612,A 0.000,B 0.000,C 90.000,E1 290.174} C_DIS
LIN {X -0.016,Y -349.790,Z 1863.605,A 0.000,B 0.000,C 90.000,E1 288.960} C_DIS
LIN {X -0.053,Y -355.136,Z 1863.600,A 0.000,B 0.000,C 90.000,E1 288.055} C_DIS
LIN {X -0.048,Y -359.894,Z 1863.595,A 0.000,B 0.000,C 90.000,E1 287.149} C_DIS
LIN {X -0.098,Y -363.899,Z 1863.590,A 0.000,B 0.000,C 90.000,E1 286.260} C_DIS
LIN {X -0.109,Y -367.236,Z 1863.585,A 0.000,B 0.000,C 90.000,E1 285.371} C_DIS
LIN {X -0.065,Y -369.130,Z 1863.582,A 0.000,B 0.000,C 90.000,E1 284.773} C_DIS
LIN {X -0.017,Y -370.634,Z 1863.579,A 0.000,B 0.000,C 90.000,E1 284.175} C_DIS
LIN {X -0.048,Y -371.751,Z 1863.575,A 0.000,B 0.000,C 90.000,E1 283.592} C_DIS
LIN {X -0.066,Y -372.507,Z 1863.572,A 0.000,B 0.000,C 90.000,E1 283.008} C_DIS
LIN {X 0.005,Y -372.807,Z 1863.569,A 0.000,B 0.000,C 90.000,E1 282.411} C_DIS
LIN {X -0.003,Y -372.710,Z 1863.566,A 0.000,B 0.000,C 90.000,E1 281.827} C_DIS
LIN {X -0.008,Y -372.176,Z 1863.563,A 0.000,B 0.000,C 90.000,E1 281.243} C_DIS
LIN {X -0.012,Y -371.210,Z 1863.559,A 0.000,B 0.000,C 90.000,E1 280.658} C_DIS
LIN {X -0.021,Y -369.870,Z 1863.556,A 0.000,B 0.000,C 90.000,E1 280.074} C_DIS
LIN {X -0.099,Y -368.145,Z 1863.553,A 0.000,B 0.000,C 90.000,E1 279.500} C_DIS
LIN {X -0.121,Y -366.158,Z 1863.549,A 0.000,B 0.000,C 90.000,E1 278.916} C_DIS
LIN {X 0.101,Y -361.709,Z 1863.543,A 0.000,B 0.000,C 90.000,E1 277.701} C_DIS
LIN {X -0.016,Y -359.207,Z 1863.540,A 0.000,B 0.000,C 90.000,E1 277.125} C_DIS
LIN {X -0.104,Y -356.273,Z 1863.536,A 0.000,B 0.000,C 90.000,E1 276.543} C_DIS
LIN {X 0.102,Y -352.789,Z 1863.533,A 0.000,B 0.000,C 90.000,E1 275.910} C_DIS
LIN {X -0.063,Y -348.721,Z 1863.530,A 0.000,B 0.000,C 90.000,E1 275.334} C_DIS
LIN {X 0.098,Y -344.043,Z 1863.526,A 0.000,B 0.000,C 90.000,E1 274.702} C_DIS
LIN {X -0.136,Y -338.606,Z 1863.523,A 0.000,B 0.000,C 90.000,E1 274.131} C_DIS
LIN {X 0.127,Y -332.786,Z 1863.520,A 0.000,B 0.000,C 90.000,E1 273.498} C_DIS
LIN {X -0.041,Y -326.625,Z 1863.516,A 0.000,B 0.000,C 90.000,E1 272.980} C_DIS
LIN {X 0.079,Y -320.334,Z 1863.514,A 0.000,B 0.000,C 90.000,E1 272.465} C_DIS
LIN {X 0.134,Y -313.572,Z 1863.511,A 0.000,B 0.000,C 90.000,E1 272.007} C_DIS
LIN {X -0.083,Y -306.853,Z 1863.509,A 0.000,B 0.000,C 90.000,E1 271.661} C_DIS
LIN {X -0.045,Y -299.499,Z 1863.507,A 0.000,B 0.000,C 90.000,E1 271.318} C_DIS
LIN {X 0.044,Y -291.875,Z 1863.506,A 0.000,B 0.000,C 90.000,E1 271.031} C_DIS
LIN {X 0.127,Y -284.195,Z 1863.505,A 0.000,B 0.000,C 90.000,E1 270.802} C_DIS
LIN {X 0.049,Y -272.595,Z 1863.503,A 0.000,B 0.000,C 90.000,E1 270.573} C_DIS
LIN {X -0.014,Y -247.682,Z 1863.501,A 0.000,B 0.000,C 90.000,E1 270.115} C_DIS
LIN {X -0.116,Y -238.598,Z 1863.500,A 0.000,B 0.000,C 90.000,E1 270.000} C_DIS
LIN {X -0.036,Y -228.330,Z 1863.499,A 0.000,B 0.000,C 90.000,E1 269.885} C_DIS
LIN {X -0.052,Y -181.535,Z 1863.499,A 0.000,B 0.000,C 90.000,E1 269.885} C_DIS
LIN {X 0.046,Y -180.904,Z 1863.474,A 0.000,B 0.000,C 90.000,E1 265.298} C_DIS
LIN {X -0.005,Y -180.250,Z 1863.465,A 0.000,B 0.000,C 90.000,E1 263.628} C_DIS
LIN {X 0.014,Y -178.740,Z 1863.441,A 0.000,B 0.000,C 90.000,E1 259.398} C_DIS
LIN {X -0.088,Y -175.788,Z 1863.413,A 0.000,B 0.000,C 90.000,E1 254.338} C_DIS
LIN {X -0.093,Y -171.971,Z 1863.384,A 0.000,B 0.000,C 90.000,E1 249.209} C_DIS
LIN {X -0.054,Y -171.372,Z 1863.380,A 0.000,B 0.000,C 90.000,E1 248.337} C_DIS
LIN {X -0.068,Y -167.619,Z 1863.356,A 0.000,B 0.000,C 90.000,E1 244.024} C_DIS
LIN {X -0.053,Y -166.269,Z 1863.346,A 0.000,B 0.000,C 90.000,E1 242.281} C_DIS
LIN {X -0.058,Y -163.021,Z 1863.327,A 0.000,B 0.000,C 90.000,E1 238.791} C_DIS
LIN {X -0.006,Y -160.948,Z 1863.312,A 0.000,B 0.000,C 90.000,E1 236.135} C_DIS
LIN {X -0.022,Y -157.704,Z 1863.292,A 0.000,B 0.000,C 90.000,E1 232.603} C_DIS
LIN {X 0.042,Y -155.744,Z 1863.277,A 0.000,B 0.000,C 90.000,E1 229.908} C_DIS
LIN {X -0.013,Y -152.001,Z 1863.252,A 0.000,B 0.000,C 90.000,E1 225.445} C_DIS
LIN {X 0.000,Y -150.247,Z 1863.237,A 0.000,B 0.000,C 90.000,E1 222.732} C_DIS
LIN {X 0.033,Y -147.004,Z 1863.212,A 0.000,B 0.000,C 90.000,E1 218.177} C_DIS
LIN {X 0.023,Y -145.588,Z 1863.197,A 0.000,B 0.000,C 90.000,E1 215.438} C_DIS
LIN {X -0.057,Y -142.976,Z 1863.171,A 0.000,B 0.000,C 90.000,E1 210.875} C_DIS
LIN {X 0.069,Y -141.603,Z 1863.151,A 0.000,B 0.000,C 90.000,E1 207.129} C_DIS
LIN {X -0.015,Y -139.424,Z 1863.115,A 0.000,B 0.000,C 90.000,E1 200.663} C_DIS
LIN {X 0.036,Y -139.152,Z 1863.104,A 0.000,B 0.000,C 90.000,E1 198.779} C_DIS
LIN {X 0.058,Y -138.345,Z 1863.058,A 0.000,B 0.000,C 90.000,E1 190.366} C_DIS
LIN {X 0.043,Y -139.484,Z 1863.006,A 0.000,B 0.000,C 90.000,E1 181.031} C_DIS
LIN {X -0.016,Y -141.082,Z 1862.975,A 0.000,B 0.000,C 90.000,E1 175.469} C_DIS
LIN {X -0.062,Y -142.458,Z 1862.959,A 0.000,B 0.000,C 90.000,E1 172.704} C_DIS
LIN {X 0.027,Y -144.702,Z 1862.934,A 0.000,B 0.000,C 90.000,E1 168.049} C_DIS
LIN {X -0.021,Y -147.298,Z 1862.913,A 0.000,B 0.000,C 90.000,E1 164.393} C_DIS
LIN {X -0.006,Y -150.617,Z 1862.888,A 0.000,B 0.000,C 90.000,E1 159.826} C_DIS
LIN {X -0.070,Y -154.092,Z 1862.868,A 0.000,B 0.000,C 90.000,E1 156.230} C_DIS
LIN {X -0.005,Y -157.515,Z 1862.848,A 0.000,B 0.000,C 90.000,E1 152.615} C_DIS
LIN {X -0.061,Y -161.747,Z 1862.828,A 0.000,B 0.000,C 90.000,E1 149.076} C_DIS
LIN {X 0.047,Y -165.940,Z 1862.808,A 0.000,B 0.000,C 90.000,E1 145.515} C_DIS
LIN {X 0.044,Y -170.930,Z 1862.789,A 0.000,B 0.000,C 90.000,E1 142.029} C_DIS
LIN {X -0.035,Y -175.799,Z 1862.770,A 0.000,B 0.000,C 90.000,E1 138.609} C_DIS
LIN {X 0.092,Y -181.406,Z 1862.751,A 0.000,B 0.000,C 90.000,E1 135.162} C_DIS
LIN {X -0.033,Y -186.907,Z 1862.732,A 0.000,B 0.000,C 90.000,E1 131.838} C_DIS
LIN {X -0.081,Y -191.487,Z 1862.719,A 0.000,B 0.000,C 90.000,E1 129.358} C_DIS
LIN {X 0.126,Y -197.349,Z 1862.700,A 0.000,B 0.000,C 90.000,E1 126.011} C_DIS
LIN {X 0.051,Y -200.625,Z 1862.691,A 0.000,B 0.000,C 90.000,E1 124.405} C_DIS
LIN {X -0.039,Y -206.508,Z 1862.673,A 0.000,B 0.000,C 90.000,E1 121.209} C_DIS
LIN {X -0.048,Y -209.798,Z 1862.664,A 0.000,B 0.000,C 90.000,E1 119.617} C_DIS
LIN {X -0.017,Y -217.158,Z 1862.643,A 0.000,B 0.000,C 90.000,E1 115.668} C_DIS
LIN {X -0.063,Y -218.784,Z 1862.638,A 0.000,B 0.000,C 90.000,E1 114.899} C_DIS
LIN {X 0.042,Y -224.090,Z 1862.621,A 0.000,B 0.000,C 90.000,E1 111.844} C_DIS
LIN {X 0.018,Y -283.809,Z 1862.621,A 0.000,B 0.000,C 90.000,E1 111.844} C_DIS
LIN {X 0.077,Y -286.455,Z 1862.621,A 0.000,B 0.000,C 90.000,E1 111.770} C_DIS
LIN {X 0.124,Y -289.647,Z 1862.620,A 0.000,B 0.000,C 90.000,E1 111.589} C_DIS
LIN {X 0.004,Y -293.205,Z 1862.618,A 0.000,B 0.000,C 90.000,E1 111.280} C_DIS
LIN {X 0.022,Y -296.804,Z 1862.615,A 0.000,B 0.000,C 90.000,E1 110.737} C_DIS
LIN {X 0.027,Y -310.094,Z 1862.602,A 0.000,B 0.000,C 90.000,E1 108.417} C_DIS
LIN {X 0.049,Y -324.750,Z 1862.590,A 0.000,B 0.000,C 90.000,E1 106.150} C_DIS
LIN {X 0.125,Y -338.497,Z 1862.579,A 0.000,B 0.000,C 90.000,E1 104.245} C_DIS
LIN {X 0.040,Y -353.435,Z 1862.569,A 0.000,B 0.000,C 90.000,E1 102.411} C_DIS
LIN {X 0.133,Y -371.841,Z 1862.558,A 0.000,B 0.000,C 90.000,E1 100.366} C_DIS
LIN {X 0.186,Y -390.723,Z 1862.547,A 0.000,B 0.000,C 90.000,E1 98.511} C_DIS
LIN {X 0.174,Y -409.947,Z 1862.538,A 0.000,B 0.000,C 90.000,E1 96.834} C_DIS
LIN {X 0.059,Y -432.337,Z 1862.528,A 0.000,B 0.000,C 90.000,E1 95.106} C_DIS
LIN {X 0.025,Y -437.993,Z 1862.526,A 0.000,B 0.000,C 90.000,E1 94.702} C_DIS
LIN {X -0.211,Y -440.544,Z 1862.525,A 0.000,B 0.000,C 90.000,E1 94.531} C_DIS
LIN {X -0.025,Y -444.162,Z 1862.523,A 0.000,B 0.000,C 90.000,E1 94.073} C_DIS
LIN {X 0.177,Y -445.653,Z 1862.521,A 0.000,B 0.000,C 90.000,E1 93.784} C_DIS
LIN {X -0.098,Y -446.775,Z 1862.520,A 0.000,B 0.000,C 90.000,E1 93.555} C_DIS
LIN {X -0.144,Y -448.129,Z 1862.517,A 0.000,B 0.000,C 90.000,E1 93.037} C_DIS
LIN {X -0.209,Y -448.498,Z 1862.514,A 0.000,B 0.000,C 90.000,E1 92.522} C_DIS
LIN {X 0.187,Y -447.941,Z 1862.511,A 0.000,B 0.000,C 90.000,E1 91.949} C_DIS
LIN {X 0.149,Y -446.375,Z 1862.508,A 0.000,B 0.000,C 90.000,E1 91.432} C_DIS
LIN {X -0.100,Y -445.134,Z 1862.507,A 0.000,B 0.000,C 90.000,E1 91.203} C_DIS
LIN {X -0.161,Y -433.662,Z 1862.496,A 0.000,B 0.000,C 90.000,E1 89.370} C_DIS
LIN {X -0.140,Y -423.666,Z 1862.487,A 0.000,B 0.000,C 90.000,E1 87.764} C_DIS
LIN {X -0.180,Y -411.882,Z 1862.477,A 0.000,B 0.000,C 90.000,E1 85.869} C_DIS
LIN {X -0.017,Y -400.005,Z 1862.466,A 0.000,B 0.000,C 90.000,E1 83.913} C_DIS
LIN {X -0.071,Y -388.050,Z 1862.455,A 0.000,B 0.000,C 90.000,E1 81.951} C_DIS
LIN {X 0.058,Y -376.141,Z 1862.444,A 0.000,B 0.000,C 90.000,E1 79.926} C_DIS
LIN {X 0.059,Y -359.558,Z 1862.428,A 0.000,B 0.000,C 90.000,E1 76.992} C_DIS
LIN {X 0.092,Y -344.030,Z 1862.411,A 0.000,B 0.000,C 90.000,E1 73.976} C_DIS
LIN {X 0.093,Y -332.083,Z 1862.397,A 0.000,B 0.000,C 90.000,E1 71.511} C_DIS
LIN {X -0.091,Y -320.398,Z 1862.383,A 0.000,B 0.000,C 90.000,E1 69.028} C_DIS
LIN {X 0.109,Y -307.821,Z 1862.367,A 0.000,B 0.000,C 90.000,E1 66.102} C_DIS
LIN {X 0.055,Y -298.269,Z 1862.355,A 0.000,B 0.000,C 90.000,E1 63.819} C_DIS
LIN {X -0.087,Y -287.557,Z 1862.340,A 0.000,B 0.000,C 90.000,E1 61.179} C_DIS
LIN {X -0.036,Y -278.143,Z 1862.327,A 0.000,B 0.000,C 90.000,E1 58.791} C_DIS
LIN {X -0.049,Y -268.683,Z 1862.313,A 0.000,B 0.000,C 90.000,E1 56.373} C_DIS
LIN {X -0.102,Y -260.494,Z 1862.301,A 0.000,B 0.000,C 90.000,E1 54.276} C_DIS
LIN {X 0.026,Y -250.888,Z 1862.287,A 0.000,B 0.000,C 90.000,E1 51.743} C_DIS
LIN {X -0.087,Y -241.342,Z 1862.273,A 0.000,B 0.000,C 90.000,E1 49.218} C_DIS
LIN {X 0.023,Y -230.653,Z 1862.257,A 0.000,B 0.000,C 90.000,E1 46.215} C_DIS
LIN {X 0.012,Y -220.459,Z 1862.240,A 0.000,B 0.000,C 90.000,E1 43.176} C_DIS
LIN {X -0.071,Y -210.835,Z 1862.223,A 0.000,B 0.000,C 90.000,E1 40.092} C_DIS
LIN {X 0.122,Y -202.061,Z 1862.205,A 0.000,B 0.000,C 90.000,E1 36.870} C_DIS
LIN {X -0.082,Y -194.117,Z 1862.187,A 0.000,B 0.000,C 90.000,E1 33.706} C_DIS
LIN {X -0.035,Y -186.906,Z 1862.169,A 0.000,B 0.000,C 90.000,E1 30.413} C_DIS
LIN {X -0.023,Y -180.379,Z 1862.150,A 0.000,B 0.000,C 90.000,E1 27.078} C_DIS
LIN {X 0.072,Y -175.956,Z 1862.136,A 0.000,B 0.000,C 90.000,E1 24.515} C_DIS
LIN {X 0.070,Y -170.806,Z 1862.117,A 0.000,B 0.000,C 90.000,E1 21.099} C_DIS
LIN {X 0.082,Y -166.410,Z 1862.098,A 0.000,B 0.000,C 90.000,E1 17.638} C_DIS
LIN {X -0.003,Y -162.813,Z 1862.079,A 0.000,B 0.000,C 90.000,E1 14.175} C_DIS
LIN {X -0.039,Y -159.168,Z 1862.054,A 0.000,B 0.000,C 90.000,E1 9.782} C_DIS
LIN {X 0.053,Y -156.628,Z 1862.028,A 0.000,B 0.000,C 90.000,E1 5.106} C_DIS
LIN {X 0.026,Y -168.753,Z 1862.028,A 0.000,B 0.000,C 90.000,E1 5.106} C_DIS
LIN {X -0.011,Y -169.983,Z 1862.028,A 0.000,B 0.000,C 90.000,E1 4.992} C_DIS
LIN {X 0.053,Y -171.966,Z 1862.025,A 0.000,B 0.000,C 90.000,E1 4.416} C_DIS
LIN {X 0.044,Y -173.648,Z 1862.020,A 0.000,B 0.000,C 90.000,E1 3.555} C_DIS
LIN {X 0.047,Y -174.835,Z 1862.015,A 0.000,B 0.000,C 90.000,E1 2.694} C_DIS
LIN {X 0.070,Y -176.615,Z 1862.005,A 0.000,B 0.000,C 90.000,E1 0.974} C_DIS
LIN {X -0.003,Y -178.500,Z 1861.993,A 0.000,B 0.000,C 90.000,E1 358.682} C_DIS
LIN {X -0.016,Y -180.852,Z 1861.974,A 0.000,B 0.000,C 90.000,E1 355.298} C_DIS
LIN {X 0.008,Y -182.433,Z 1861.960,A 0.000,B 0.000,C 90.000,E1 352.761} C_DIS
LIN {X 0.026,Y -184.523,Z 1861.941,A 0.000,B 0.000,C 90.000,E1 349.398} C_DIS
LIN {X 0.010,Y -186.633,Z 1861.923,A 0.000,B 0.000,C 90.000,E1 346.061} C_DIS
LIN {X 0.045,Y -188.745,Z 1861.904,A 0.000,B 0.000,C 90.000,E1 342.725} C_DIS
LIN {X -0.054,Y -190.861,Z 1861.886,A 0.000,B 0.000,C 90.000,E1 339.444} C_DIS
LIN {X 0.026,Y -193.662,Z 1861.863,A 0.000,B 0.000,C 90.000,E1 335.305} C_DIS
LIN {X 0.048,Y -196.141,Z 1861.845,A 0.000,B 0.000,C 90.000,E1 332.025} C_DIS
LIN {X -0.023,Y -198.648,Z 1861.827,A 0.000,B 0.000,C 90.000,E1 328.791} C_DIS
LIN {X -0.102,Y -201.946,Z 1861.804,A 0.000,B 0.000,C 90.000,E1 324.769} C_DIS
LIN {X 0.012,Y -205.732,Z 1861.782,A 0.000,B 0.000,C 90.000,E1 320.723} C_DIS
LIN {X -0.049,Y -209.328,Z 1861.764,A 0.000,B 0.000,C 90.000,E1 317.553} C_DIS
LIN {X 0.013,Y -212.796,Z 1861.751,A 0.000,B 0.000,C 90.000,E1 315.162} C_DIS
LIN {X -0.112,Y -215.643,Z 1861.742,A 0.000,B 0.000,C 90.000,E1 313.623} C_DIS
LIN {X -0.051,Y -219.094,Z 1861.734,A 0.000,B 0.000,C 90.000,E1 312.043} C_DIS
LIN {X 0.009,Y -222.252,Z 1861.727,A 0.000,B 0.000,C 90.000,E1 310.862} C_DIS
LIN {X -0.065,Y -225.933,Z 1861.721,A 0.000,B 0.000,C 90.000,E1 309.725} C_DIS
LIN {X 0.072,Y -230.076,Z 1861.714,A 0.000,B 0.000,C 90.000,E1 308.543} C_DIS
LIN {X 0.030,Y -237.995,Z 1861.704,A 0.000,B 0.000,C 90.000,E1 306.664} C_DIS
LIN {X -0.028,Y -246.837,Z 1861.693,A 0.000,B 0.000,C 90.000,E1 304.818} C_DIS
LIN {X -0.004,Y -258.477,Z 1861.681,A 0.000,B 0.000,C 90.000,E1 302.625} C_DIS
LIN {X -0.034,Y -269.172,Z 1861.671,A 0.000,B 0.000,C 90.000,E1 300.846} C_DIS
LIN {X -0.032,Y -285.281,Z 1861.658,A 0.000,B 0.000,C 90.000,E1 298.409} C_DIS
LIN {X 0.068,Y -296.895,Z 1861.648,A 0.000,B 0.000,C 90.000,E1 296.693} C_DIS
LIN {X -0.005,Y -310.831,Z 1861.637,A 0.000,B 0.000,C 90.000,E1 294.719} C_DIS
LIN {X 0.120,Y -322.214,Z 1861.628,A 0.000,B 0.000,C 90.000,E1 293.078} C_DIS
LIN {X -0.140,Y -333.503,Z 1861.620,A 0.000,B 0.000,C 90.000,E1 291.535} C_DIS
LIN {X 0.095,Y -342.072,Z 1861.613,A 0.000,B 0.000,C 90.000,E1 290.248} C_DIS
LIN {X 0.002,Y -349.974,Z 1861.606,A 0.000,B 0.000,C 90.000,E1 289.033} C_DIS
LIN {X 0.003,Y -357.071,Z 1861.599,A 0.000,B 0.000,C 90.000,E1 287.819} C_DIS
LIN {X 0.033,Y -361.616,Z 1861.594,A 0.000,B 0.000,C 90.000,E1 286.913} C_DIS
LIN {X -0.002,Y -365.440,Z 1861.589,A 0.000,B 0.000,C 90.000,E1 286.024} C_DIS
LIN {X 0.032,Y -367.591,Z 1861.586,A 0.000,B 0.000,C 90.000,E1 285.426} C_DIS
LIN {X 0.077,Y -369.483,Z 1861.582,A 0.000,B 0.000,C 90.000,E1 284.828} C_DIS
LIN {X 0.036,Y -371.021,Z 1861.579,A 0.000,B 0.000,C 90.000,E1 284.245} C_DIS
LIN {X 0.098,Y -372.176,Z 1861.576,A 0.000,B 0.000,C 90.000,E1 283.647} C_DIS
LIN {X 0.081,Y -372.955,Z 1861.573,A 0.000,B 0.000,C 90.000,E1 283.063} C_DIS
LIN {X 0.074,Y -373.300,Z 1861.569,A 0.000,B 0.000,C 90.000,E1 282.479} C_DIS
LIN {X 0.072,Y -373.229,Z 1861.566,A 0.000,B 0.000,C 90.000,E1 281.895} C_DIS
LIN {X 0.146,Y -372.714,Z 1861.563,A 0.000,B 0.000,C 90.000,E1 281.299} C_DIS
LIN {X 0.074,Y -371.778,Z 1861.560,A 0.000,B 0.000,C 90.000,E1 280.725} C_DIS
LIN {X 0.071,Y -370.425,Z 1861.556,A 0.000,B 0.000,C 90.000,E1 280.141} C_DIS
LIN {X 0.060,Y -368.704,Z 1861.553,A 0.000,B 0.000,C 90.000,E1 279.557} C_DIS
LIN {X -0.047,Y -364.498,Z 1861.547,A 0.000,B 0.000,C 90.000,E1 278.398} C_DIS
LIN {X -0.174,Y -361.052,Z 1861.542,A 0.000,B 0.000,C 90.000,E1 277.530} C_DIS
LIN {X 0.108,Y -358.405,Z 1861.538,A 0.000,B 0.000,C 90.000,E1 276.891} C_DIS
LIN {X -0.028,Y -355.322,Z 1861.535,A 0.000,B 0.000,C 90.000,E1 276.315} C_DIS
LIN {X 0.173,Y -351.640,Z 1861.532,A 0.000,B 0.000,C 90.000,E1 275.682} C_DIS
LIN {X 0.003,Y -347.326,Z 1861.528,A 0.000,B 0.000,C 90.000,E1 275.106} C_DIS
LIN {X 0.155,Y -342.368,Z 1861.525,A 0.000,B 0.000,C 90.000,E1 274.473} C_DIS
LIN {X -0.003,Y -336.797,Z 1861.522,A 0.000,B 0.000,C 90.000,E1 273.898} C_DIS
LIN {X 0.003,Y -330.833,Z 1861.518,A 0.000,B 0.000,C 90.000,E1 273.326} C_DIS
LIN {X -0.032,Y -324.657,Z 1861.516,A 0.000,B 0.000,C 90.000,E1 272.808} C_DIS
LIN {X -0.138,Y -318.161,Z 1861.513,A 0.000,B 0.000,C 90.000,E1 272.350} C_DIS
LIN {X 0.034,Y -311.404,Z 1861.510,A 0.000,B 0.000,C 90.000,E1 271.892} C_DIS
LIN {X -0.109,Y -304.464,Z 1861.508,A 0.000,B 0.000,C 90.000,E1 271.547} C_DIS
LIN {X 0.065,Y -296.891,Z 1861.507,A 0.000,B 0.000,C 90.000,E1 271.203} C_DIS
LIN {X -0.031,Y -289.341,Z 1861.505,A 0.000,B 0.000,C 90.000,E1 270.974} C_DIS
LIN {X -0.006,Y -277.652,Z 1861.504,A 0.000,B 0.000,C 90.000,E1 270.688} C_DIS
LIN {X 0.053,Y -245.093,Z 1861.500,A 0.000,B 0.000,C 90.000,E1 270.057} C_DIS
LIN {X 0.090,Y -232.270,Z 1861.500,A 0.000,B 0.000,C 90.000,E1 269.885} C_DIS
LIN {X -0.002,Y -227.983,Z 1861.499,A 0.000,B 0.000,C 90.000,E1 269.885} C_DIS
LIN {X -0.026,Y -181.537,Z 1861.499,A 0.000,B 0.000,C 90.000,E1 269.885} C_DIS
LIN {X -0.085,Y -180.905,Z 1861.474,A 0.000,B 0.000,C 90.000,E1 265.355} C_DIS
LIN {X -0.011,Y -180.668,Z 1861.469,A 0.000,B 0.000,C 90.000,E1 264.489} C_DIS
LIN {X 0.063,Y -178.749,Z 1861.441,A 0.000,B 0.000,C 90.000,E1 259.398} C_DIS
LIN {X -0.039,Y -175.797,Z 1861.413,A 0.000,B 0.000,C 90.000,E1 254.338} C_DIS
LIN {X -0.044,Y -171.982,Z 1861.384,A 0.000,B 0.000,C 90.000,E1 249.209} C_DIS
LIN {X -0.005,Y -171.387,Z 1861.380,A 0.000,B 0.000,C 90.000,E1 248.337} C_DIS
LIN {X -0.020,Y -167.631,Z 1861.356,A 0.000,B 0.000,C 90.000,E1 244.024} C_DIS
LIN {X -0.005,Y -166.286,Z 1861.346,A 0.000,B 0.000,C 90.000,E1 242.281} C_DIS
LIN {X -0.011,Y -163.034,Z 1861.327,A 0.000,B 0.000,C 90.000,E1 238.791} C_DIS
LIN {X 0.040,Y -160.965,Z 1861.312,A 0.000,B 0.000,C 90.000,E1 236.135} C_DIS
LIN {X -0.071,Y -157.717,Z 1861.292,A 0.000,B 0.000,C 90.000,E1 232.637} C_DIS
LIN {X 0.087,Y -155.757,Z 1861.277,A 0.000,B 0.000,C 90.000,E1 229.908} C_DIS
LIN {X -0.076,Y -152.012,Z 1861.253,A 0.000,B 0.000,C 90.000,E1 225.486} C_DIS
LIN {X -0.058,Y -150.259,Z 1861.238,A 0.000,B 0.000,C 90.000,E1 222.771} C_DIS
LIN {X 0.076,Y -147.014,Z 1861.212,A 0.000,B 0.000,C 90.000,E1 218.177} C_DIS
LIN {X -0.018,Y -145.597,Z 1861.197,A 0.000,B 0.000,C 90.000,E1 215.471} C_DIS
LIN {X -0.014,Y -142.984,Z 1861.172,A 0.000,B 0.000,C 90.000,E1 210.875} C_DIS
LIN {X -0.014,Y -141.611,Z 1861.151,A 0.000,B 0.000,C 90.000,E1 207.180} C_DIS
LIN {X 0.027,Y -139.427,Z 1861.115,A 0.000,B 0.000,C 90.000,E1 200.663} C_DIS
LIN {X 0.078,Y -139.157,Z 1861.104,A 0.000,B 0.000,C 90.000,E1 198.779} C_DIS
LIN {X -0.036,Y -138.343,Z 1861.058,A 0.000,B 0.000,C 90.000,E1 190.423} C_DIS
LIN {X -0.054,Y -139.482,Z 1861.006,A 0.000,B 0.000,C 90.000,E1 181.088} C_DIS
LIN {X 0.027,Y -141.075,Z 1860.975,A 0.000,B 0.000,C 90.000,E1 175.469} C_DIS
LIN {X -0.019,Y -142.450,Z 1860.959,A 0.000,B 0.000,C 90.000,E1 172.704} C_DIS
LIN {X 0.071,Y -144.691,Z 1860.934,A 0.000,B 0.000,C 90.000,E1 168.049} C_DIS
LIN {X 0.024,Y -147.284,Z 1860.913,A 0.000,B 0.000,C 90.000,E1 164.393} C_DIS
LIN {X 0.039,Y -150.603,Z 1860.888,A 0.000,B 0.000,C 90.000,E1 159.826} C_DIS
LIN {X -0.025,Y -154.077,Z 1860.868,A 0.000,B 0.000,C 90.000,E1 156.230} C_DIS
LIN {X 0.041,Y -157.497,Z 1860.848,A 0.000,B 0.000,C 90.000,E1 152.615} C_DIS
LIN {X -0.013,Y -161.726,Z 1860.828,A 0.000,B 0.000,C 90.000,E1 149.076} C_DIS
LIN {X 0.000,Y -165.919,Z 1860.809,A 0.000,B 0.000,C 90.000,E1 145.548} C_DIS
LIN {X -0.013,Y -170.905,Z 1860.789,A 0.000,B 0.000,C 90.000,E1 142.065} C_DIS
LIN {X 0.014,Y -175.774,Z 1860.770,A 0.000,B 0.000,C 90.000,E1 138.609} C_DIS
LIN {X 0.015,Y -181.383,Z 1860.751,A 0.000,B 0.000,C 90.000,E1 135.202} C_DIS
LIN {X 0.018,Y -186.879,Z 1860.732,A 0.000,B 0.000,C 90.000,E1 131.838} C_DIS
LIN {X -0.029,Y -191.462,Z 1860.719,A 0.000,B 0.000,C 90.000,E1 129.358} C_DIS
LIN {X -0.097,Y -197.319,Z 1860.700,A 0.000,B 0.000,C 90.000,E1 126.091} C_DIS
LIN {X 0.104,Y -200.596,Z 1860.691,A 0.000,B 0.000,C 90.000,E1 124.405} C_DIS
LIN {X 0.015,Y -206.479,Z 1860.673,A 0.000,B 0.000,C 90.000,E1 121.209} C_DIS
LIN {X 0.007,Y -209.766,Z 1860.665,A 0.000,B 0.000,C 90.000,E1 119.617} C_DIS
LIN {X 0.038,Y -217.128,Z 1860.643,A 0.000,B 0.000,C 90.000,E1 115.668} C_DIS
LIN {X -0.007,Y -218.754,Z 1860.638,A 0.000,B 0.000,C 90.000,E1 114.899} C_DIS
LIN {X 0.066,Y -224.079,Z 1860.621,A 0.000,B 0.000,C 90.000,E1 111.844} C_DIS
LIN {X 0.048,Y -283.214,Z 1860.621,A 0.000,B 0.000,C 90.000,E1 111.844} C_DIS
LIN {X 0.043,Y -286.081,Z 1860.621,A 0.000,B 0.000,C 90.000,E1 111.791} C_DIS
LIN {X 0.012,Y -288.883,Z 1860.620,A 0.000,B 0.000,C 90.000,E1 111.663} C_DIS
LIN {X 0.069,Y -292.435,Z 1860.619,A 0.000,B 0.000,C 90.000,E1 111.354} C_DIS
LIN {X 0.051,Y -296.060,Z 1860.616,A 0.000,B 0.000,C 90.000,E1 110.865} C_DIS
LIN {X 0.045,Y -309.303,Z 1860.603,A 0.000,B 0.000,C 90.000,E1 108.544} C_DIS
LIN {X 0.144,Y -323.876,Z 1860.590,A 0.000,B 0.000,C 90.000,E1 106.260} C_DIS
LIN {X -0.126,Y -337.549,Z 1860.580,A 0.000,B 0.000,C 90.000,E1 104.411} C_DIS
LIN {X 0.020,Y -352.405,Z 1860.570,A 0.000,B 0.000,C 90.000,E1 102.535} C_DIS
LIN {X 0.046,Y -370.785,Z 1860.558,A 0.000,B 0.000,C 90.000,E1 100.489} C_DIS
LIN {X 0.094,Y -389.644,Z 1860.548,A 0.000,B 0.000,C 90.000,E1 98.624} C_DIS
LIN {X 0.012,Y -408.847,Z 1860.539,A 0.000,B 0.000,C 90.000,E1 96.947} C_DIS
LIN {X -0.182,Y -431.217,Z 1860.529,A 0.000,B 0.000,C 90.000,E1 95.220} C_DIS
LIN {X -0.042,Y -439.633,Z 1860.526,A 0.000,B 0.000,C 90.000,E1 94.588} C_DIS
LIN {X -0.117,Y -443.452,Z 1860.523,A 0.000,B 0.000,C 90.000,E1 94.188} C_DIS
LIN {X 0.081,Y -445.115,Z 1860.522,A 0.000,B 0.000,C 90.000,E1 93.898} C_DIS
LIN {X -0.196,Y -446.370,Z 1860.520,A 0.000,B 0.000,C 90.000,E1 93.669} C_DIS
LIN {X 0.201,Y -447.936,Z 1860.517,A 0.000,B 0.000,C 90.000,E1 93.094} C_DIS
LIN {X 0.135,Y -448.484,Z 1860.514,A 0.000,B 0.000,C 90.000,E1 92.579} C_DIS
LIN {X 0.080,Y -448.107,Z 1860.511,A 0.000,B 0.000,C 90.000,E1 92.064} C_DIS
LIN {X 0.043,Y -446.749,Z 1860.509,A 0.000,B 0.000,C 90.000,E1 91.547} C_DIS
LIN {X -0.206,Y -445.638,Z 1860.507,A 0.000,B 0.000,C 90.000,E1 91.318} C_DIS
LIN {X 0.180,Y -442.502,Z 1860.504,A 0.000,B 0.000,C 90.000,E1 90.745} C_DIS
LIN {X 0.205,Y -429.335,Z 1860.493,A 0.000,B 0.000,C 90.000,E1 88.625} C_DIS
LIN {X -0.147,Y -417.559,Z 1860.482,A 0.000,B 0.000,C 90.000,E1 86.788} C_DIS
LIN {X 0.094,Y -405.754,Z 1860.471,A 0.000,B 0.000,C 90.000,E1 84.837} C_DIS
LIN {X 0.158,Y -393.821,Z 1860.461,A 0.000,B 0.000,C 90.000,E1 82.875} C_DIS
LIN {X 0.026,Y -381.874,Z 1860.449,A 0.000,B 0.000,C 90.000,E1 80.905} C_DIS
LIN {X 0.082,Y -368.338,Z 1860.437,A 0.000,B 0.000,C 90.000,E1 78.578} C_DIS
LIN {X -0.105,Y -350.700,Z 1860.418,A 0.000,B 0.000,C 90.000,E1 75.338} C_DIS
LIN {X -0.131,Y -338.577,Z 1860.405,A 0.000,B 0.000,C 90.000,E1 72.906} C_DIS
LIN {X 0.155,Y -326.744,Z 1860.391,A 0.000,B 0.000,C 90.000,E1 70.369} C_DIS
LIN {X -0.077,Y -312.465,Z 1860.373,A 0.000,B 0.000,C 90.000,E1 67.230} C_DIS
LIN {X 0.139,Y -301.518,Z 1860.359,A 0.000,B 0.000,C 90.000,E1 64.588} C_DIS
LIN {X -0.074,Y -289.356,Z 1860.342,A 0.000,B 0.000,C 90.000,E1 61.641} C_DIS
LIN {X 0.051,Y -281.325,Z 1860.331,A 0.000,B 0.000,C 90.000,E1 59.587} C_DIS
LIN {X 0.021,Y -273.237,Z 1860.320,A 0.000,B 0.000,C 90.000,E1 57.533} C_DIS
LIN {X -0.100,Y -265.124,Z 1860.308,A 0.000,B 0.000,C 90.000,E1 55.468} C_DIS
LIN {X -0.020,Y -255.512,Z 1860.294,A 0.000,B 0.000,C 90.000,E1 52.970} C_DIS
LIN {X -0.001,Y -245.921,Z 1860.280,A 0.000,B 0.000,C 90.000,E1 50.436} C_DIS
LIN {X -0.070,Y -236.451,Z 1860.266,A 0.000,B 0.000,C 90.000,E1 47.877} C_DIS
LIN {X -0.005,Y -224.708,Z 1860.247,A 0.000,B 0.000,C 90.000,E1 44.474} C_DIS
LIN {X 0.065,Y -213.606,Z 1860.228,A 0.000,B 0.000,C 90.000,E1 40.987} C_DIS
LIN {X -0.009,Y -204.550,Z 1860.210,A 0.000,B 0.000,C 90.000,E1 37.855} C_DIS
LIN {X -0.040,Y -196.401,Z 1860.193,A 0.000,B 0.000,C 90.000,E1 34.659} C_DIS
LIN {X -0.006,Y -188.957,Z 1860.174,A 0.000,B 0.000,C 90.000,E1 31.386} C_DIS
LIN {X -0.113,Y -182.238,Z 1860.156,A 0.000,B 0.000,C 90.000,E1 28.103} C_DIS
LIN {X 0.015,Y -176.215,Z 1860.137,A 0.000,B 0.000,C 90.000,E1 24.695} C_DIS
LIN {X 0.018,Y -171.029,Z 1860.118,A 0.000,B 0.000,C 90.000,E1 21.280} C_DIS
LIN {X 0.036,Y -166.595,Z 1860.099,A 0.000,B 0.000,C 90.000,E1 17.819} C_DIS
LIN {X -0.042,Y -162.961,Z 1860.080,A 0.000,B 0.000,C 90.000,E1 14.356} C_DIS
LIN {X -0.069,Y -159.277,Z 1860.055,A 0.000,B 0.000,C 90.000,E1 9.962} C_DIS
LIN {X -0.065,Y -158.510,Z 1860.049,A 0.000,B 0.000,C 90.000,E1 8.803} C_DIS
LIN {X -0.081,Y -158.772,Z 1860.049,A 0.000,B 0.000,C 90.000,E1 8.803} C_DIS
LIN {X -0.047,Y -170.574,Z 1860.047,A 0.000,B 0.000,C 90.000,E1 8.568} C_DIS
LIN {X 0.074,Y -171.536,Z 1860.047,A 0.000,B 0.000,C 90.000,E1 8.398} C_DIS
LIN {X 0.004,Y -172.562,Z 1860.045,A 0.000,B 0.000,C 90.000,E1 8.163} C_DIS
LIN {X 0.021,Y -174.415,Z 1860.041,A 0.000,B 0.000,C 90.000,E1 7.296} C_DIS
LIN {X 0.043,Y -175.559,Z 1860.036,A 0.000,B 0.000,C 90.000,E1 6.429} C_DIS
LIN {X -0.078,Y -177.144,Z 1860.026,A 0.000,B 0.000,C 90.000,E1 4.759} C_DIS
LIN {X 0.013,Y -178.888,Z 1860.012,A 0.000,B 0.000,C 90.000,E1 2.178} C_DIS
LIN {X -0.033,Y -180.373,Z 1859.997,A 0.000,B 0.000,C 90.000,E1 359.542} C_DIS
LIN {X -0.006,Y -182.124,Z 1859.979,A 0.000,B 0.000,C 90.000,E1 356.159} C_DIS
LIN {X -0.069,Y -183.838,Z 1859.960,A 0.000,B 0.000,C 90.000,E1 352.818} C_DIS
LIN {X -0.016,Y -185.586,Z 1859.941,A 0.000,B 0.000,C 90.000,E1 349.454} C_DIS
LIN {X -0.006,Y -187.419,Z 1859.923,A 0.000,B 0.000,C 90.000,E1 346.117} C_DIS
LIN {X 0.051,Y -189.283,Z 1859.904,A 0.000,B 0.000,C 90.000,E1 342.779} C_DIS
LIN {X -0.098,Y -191.179,Z 1859.886,A 0.000,B 0.000,C 90.000,E1 339.518} C_DIS
LIN {X 0.062,Y -193.718,Z 1859.863,A 0.000,B 0.000,C 90.000,E1 335.357} C_DIS
LIN {X -0.002,Y -195.988,Z 1859.845,A 0.000,B 0.000,C 90.000,E1 332.103} C_DIS
LIN {X -0.032,Y -199.001,Z 1859.822,A 0.000,B 0.000,C 90.000,E1 328.043} C_DIS
LIN {X 0.015,Y -202.397,Z 1859.800,A 0.000,B 0.000,C 90.000,E1 323.989} C_DIS
LIN {X -0.019,Y -206.340,Z 1859.778,A 0.000,B 0.000,C 90.000,E1 319.989} C_DIS
LIN {X 0.071,Y -210.207,Z 1859.760,A 0.000,B 0.000,C 90.000,E1 316.782} C_DIS
LIN {X 0.000,Y -213.992,Z 1859.747,A 0.000,B 0.000,C 90.000,E1 314.433} C_DIS
LIN {X 0.044,Y -217.142,Z 1859.738,A 0.000,B 0.000,C 90.000,E1 312.852} C_DIS
LIN {X -0.020,Y -220.990,Z 1859.729,A 0.000,B 0.000,C 90.000,E1 311.310} C_DIS
LIN {X -0.030,Y -225.797,Z 1859.721,A 0.000,B 0.000,C 90.000,E1 309.769} C_DIS
LIN {X -0.097,Y -231.470,Z 1859.712,A 0.000,B 0.000,C 90.000,E1 308.257} C_DIS
LIN {X -0.118,Y -239.577,Z 1859.702,A 0.000,B 0.000,C 90.000,E1 306.377} C_DIS
LIN {X 0.043,Y -250.519,Z 1859.690,A 0.000,B 0.000,C 90.000,E1 304.119} C_DIS
LIN {X 0.003,Y -262.575,Z 1859.677,A 0.000,B 0.000,C 90.000,E1 301.957} C_DIS
LIN {X -0.060,Y -280.609,Z 1859.662,A 0.000,B 0.000,C 90.000,E1 299.155} C_DIS
LIN {X 0.085,Y -294.611,Z 1859.651,A 0.000,B 0.000,C 90.000,E1 297.078} C_DIS
LIN {X 0.101,Y -308.575,Z 1859.639,A 0.000,B 0.000,C 90.000,E1 295.079} C_DIS
LIN {X 0.133,Y -317.808,Z 1859.632,A 0.000,B 0.000,C 90.000,E1 293.770} C_DIS
LIN {X -0.108,Y -331.470,Z 1859.622,A 0.000,B 0.000,C 90.000,E1 291.897} C_DIS
LIN {X 0.098,Y -340.219,Z 1859.615,A 0.000,B 0.000,C 90.000,E1 290.610} C_DIS
LIN {X -0.020,Y -348.365,Z 1859.608,A 0.000,B 0.000,C 90.000,E1 289.396} C_DIS
LIN {X -0.074,Y -353.939,Z 1859.603,A 0.000,B 0.000,C 90.000,E1 288.489} C_DIS
LIN {X -0.071,Y -359.055,Z 1859.598,A 0.000,B 0.000,C 90.000,E1 287.583} C_DIS
LIN {X -0.026,Y -363.375,Z 1859.593,A 0.000,B 0.000,C 90.000,E1 286.677} C_DIS
LIN {X -0.038,Y -366.954,Z 1859.588,A 0.000,B 0.000,C 90.000,E1 285.788} C_DIS
LIN {X -0.019,Y -369.943,Z 1859.583,A 0.000,B 0.000,C 90.000,E1 284.898} C_DIS
LIN {X 0.036,Y -371.453,Z 1859.579,A 0.000,B 0.000,C 90.000,E1 284.300} C_DIS
LIN {X 0.012,Y -372.649,Z 1859.576,A 0.000,B 0.000,C 90.000,E1 283.716} C_DIS
LIN {X 0.085,Y -373.443,Z 1859.573,A 0.000,B 0.000,C 90.000,E1 283.119} C_DIS
LIN {X 0.080,Y -373.781,Z 1859.570,A 0.000,B 0.000,C 90.000,E1 282.535} C_DIS
LIN {X 0.081,Y -373.717,Z 1859.566,A 0.000,B 0.000,C 90.000,E1 281.951} C_DIS
LIN {X 0.084,Y -373.247,Z 1859.563,A 0.000,B 0.000,C 90.000,E1 281.366} C_DIS
LIN {X 0.087,Y -372.325,Z 1859.560,A 0.000,B 0.000,C 90.000,E1 280.782} C_DIS
LIN {X 0.086,Y -370.900,Z 1859.557,A 0.000,B 0.000,C 90.000,E1 280.197} C_DIS
LIN {X 0.078,Y -369.189,Z 1859.553,A 0.000,B 0.000,C 90.000,E1 279.613} C_DIS
LIN {X -0.026,Y -364.926,Z 1859.547,A 0.000,B 0.000,C 90.000,E1 278.454} C_DIS
LIN {X -0.150,Y -361.511,Z 1859.542,A 0.000,B 0.000,C 90.000,E1 277.587} C_DIS
LIN {X 0.135,Y -358.911,Z 1859.539,A 0.000,B 0.000,C 90.000,E1 276.947} C_DIS
LIN {X 0.001,Y -355.865,Z 1859.535,A 0.000,B 0.000,C 90.000,E1 276.372} C_DIS
LIN {X -0.145,Y -352.304,Z 1859.532,A 0.000,B 0.000,C 90.000,E1 275.796} C_DIS
